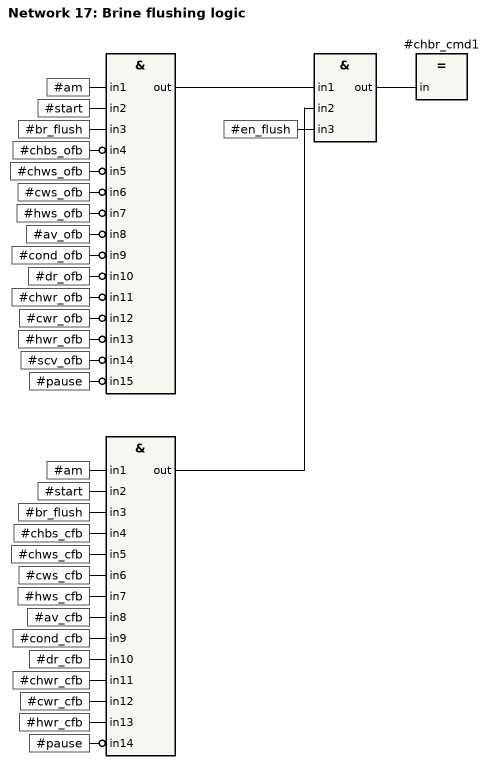
   #chbr_cmd1 := #am AND #start AND #br_flush AND NOT #chbs_ofb AND NOT #chws_ofb AND NOT #cws_ofb AND NOT #hws_ofb AND NOT #av_ofb AND NOT #cond_ofb AND NOT #dr_ofb AND NOT #chwr_ofb AND NOT #cwr_ofb AND NOT #hwr_ofb AND NOT #scv_ofb AND NOT #pause AND #am AND #start AND #br_flush AND #chbs_cfb AND #chws_cfb AND #cws_cfb AND #hws_cfb AND #av_cfb AND #cond_cfb AND #dr_cfb AND #chwr_cfb AND #cwr_cfb AND #hwr_cfb AND NOT #pause AND #en_flush;
END_REGION

REGION Network 18: Steam flushing logic
   // Steam flushing logic
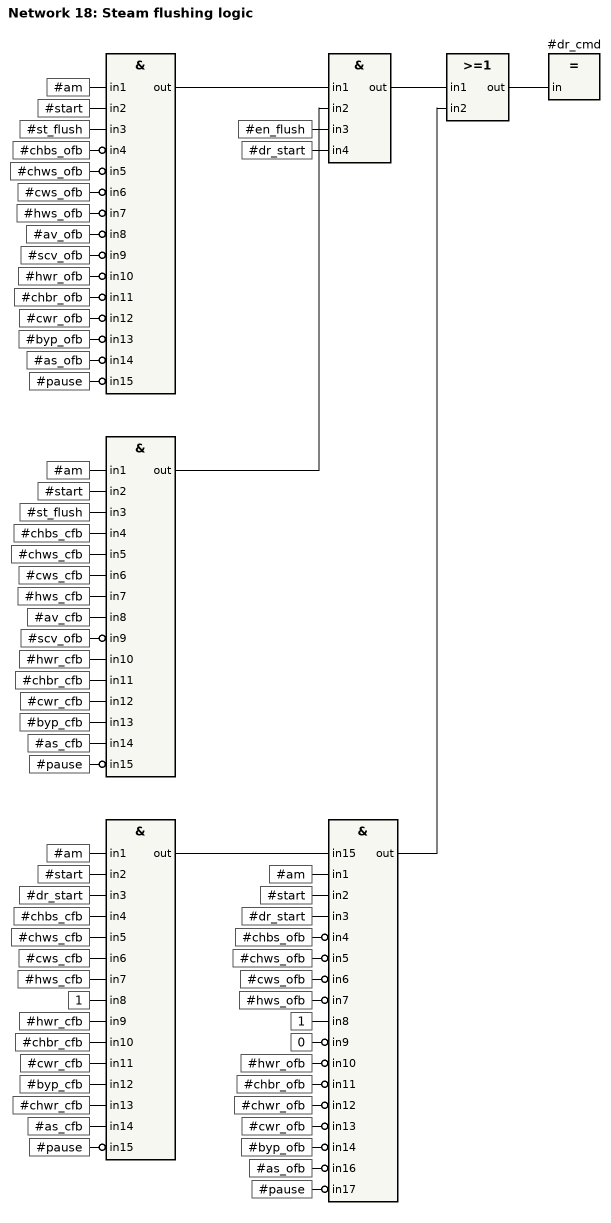
   #dr_cmd := (#am AND #start AND #st_flush AND NOT #chbs_ofb AND NOT #chws_ofb AND NOT #cws_ofb AND NOT #hws_ofb AND NOT #av_ofb AND NOT #scv_ofb AND NOT #hwr_ofb AND NOT #chbr_ofb AND NOT #cwr_ofb AND NOT #byp_ofb AND NOT #as_ofb AND NOT #pause AND #am AND #start AND #st_flush AND #chbs_cfb AND #chws_cfb AND #cws_cfb AND #hws_cfb AND #av_cfb AND NOT #scv_ofb AND #hwr_cfb AND #chbr_cfb AND #cwr_cfb AND #byp_cfb AND #as_cfb AND NOT #pause AND #en_flush AND #dr_start) OR (#am AND #start AND #dr_start AND #chbs_cfb AND #chws_cfb AND #cws_cfb AND #hws_cfb AND 1 AND #hwr_cfb AND #chbr_cfb AND #cwr_cfb AND #byp_cfb AND #chwr_cfb AND #as_cfb AND NOT #pause AND #am AND #start AND #dr_start AND NOT #chbs_ofb AND NOT #chws_ofb AND NOT #cws_ofb AND NOT #hws_ofb AND 1 AND NOT 0 AND NOT #hwr_ofb AND NOT #chbr_ofb AND NOT #chwr_ofb AND NOT #cwr_ofb AND NOT #byp_ofb AND NOT #as_ofb AND NOT #pause);
END_REGION

REGION Network 19: chw flushing logic
   // chw flushing logic
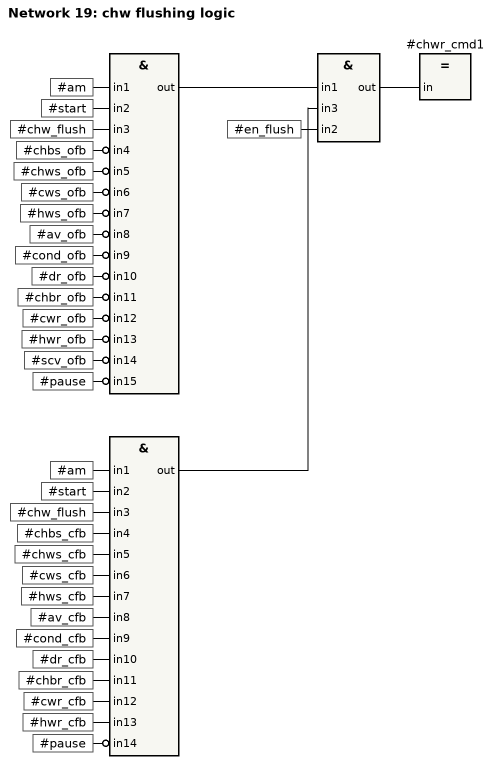
   #chwr_cmd1 := #am AND #start AND #chw_flush AND NOT #chbs_ofb AND NOT #chws_ofb AND NOT #cws_ofb AND NOT #hws_ofb AND NOT #av_ofb AND NOT #cond_ofb AND NOT #dr_ofb AND NOT #chbr_ofb AND NOT #cwr_ofb AND NOT #hwr_ofb AND NOT #scv_ofb AND NOT #pause AND #am AND #start AND #chw_flush AND #chbs_cfb AND #chws_cfb AND #cws_cfb AND #hws_cfb AND #av_cfb AND #cond_cfb AND #dr_cfb AND #chbr_cfb AND #cwr_cfb AND #hwr_cfb AND NOT #pause AND #en_flush;
END_REGION

REGION Network 20: air supply and bypass open logic
   // air supply and bypass open logic
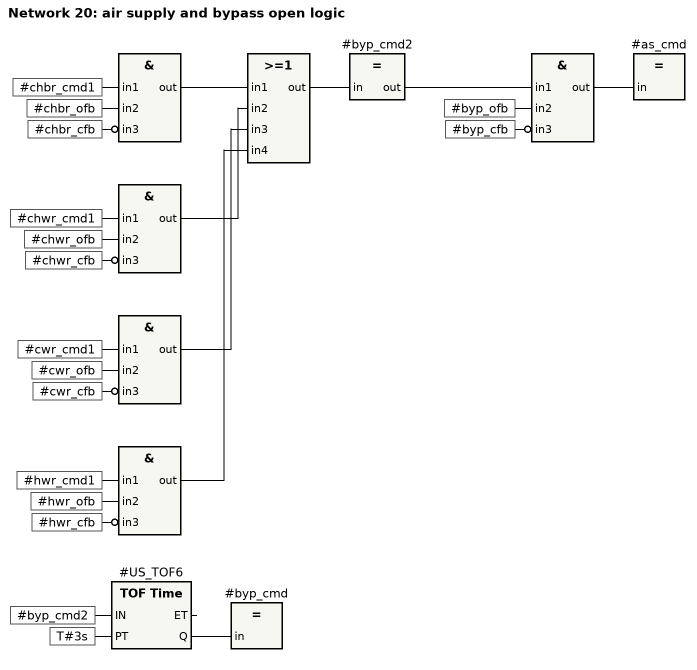
   #byp_cmd2 := (#chbr_cmd1 AND #chbr_ofb AND NOT #chbr_cfb) OR (#chwr_cmd1 AND #chwr_ofb AND NOT #chwr_cfb) OR (#cwr_cmd1 AND #cwr_ofb AND NOT #cwr_cfb) OR (#hwr_cmd1 AND #hwr_ofb AND NOT #hwr_cfb);
   #as_cmd := #byp_cmd2 AND #byp_ofb AND NOT #byp_cfb;
   #US_TOF6(IN := #byp_cmd2, PT := T#3s);   // TOF
   #byp_cmd := #US_TOF6.Q;
END_REGION

REGION Network 21: CW flushing logic
   // CW flushing logic
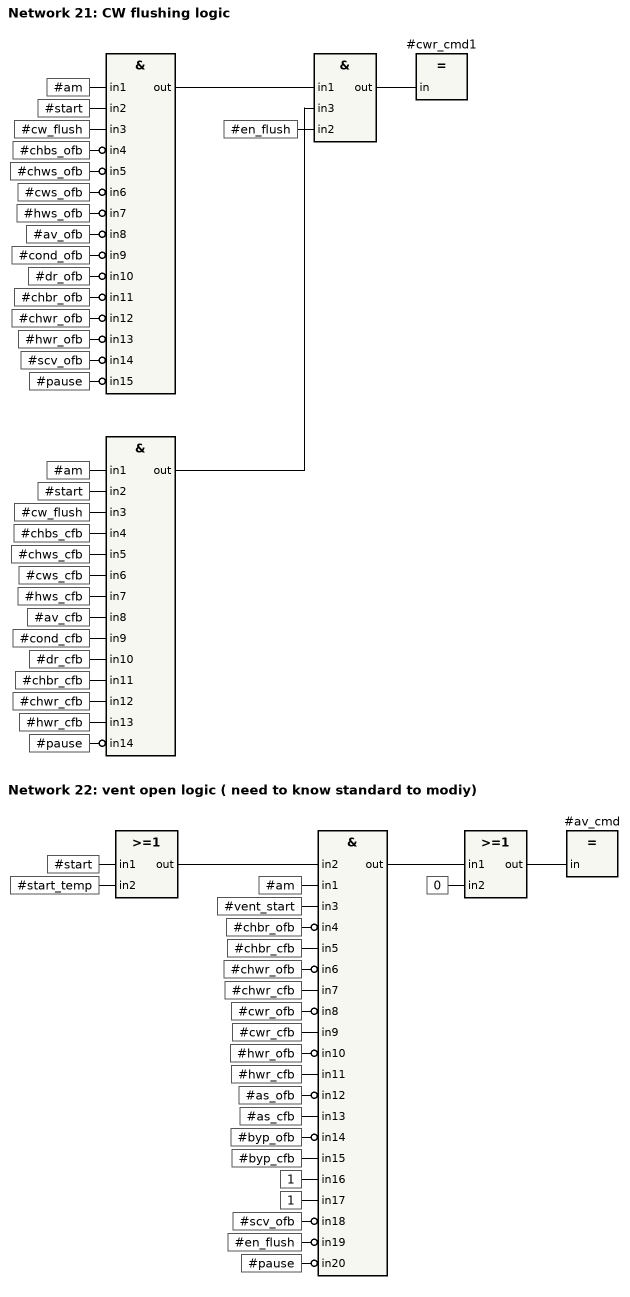
   #cwr_cmd1 := #am AND #start AND #cw_flush AND NOT #chbs_ofb AND NOT #chws_ofb AND NOT #cws_ofb AND NOT #hws_ofb AND NOT #av_ofb AND NOT #cond_ofb AND NOT #dr_ofb AND NOT #chbr_ofb AND NOT #chwr_ofb AND NOT #hwr_ofb AND NOT #scv_ofb AND NOT #pause AND #am AND #start AND #cw_flush AND #chbs_cfb AND #chws_cfb AND #cws_cfb AND #hws_cfb AND #av_cfb AND #cond_cfb AND #dr_cfb AND #chbr_cfb AND #chwr_cfb AND #hwr_cfb AND NOT #pause AND #en_flush;
END_REGION

REGION Network 22: vent open logic ( need to know standard to modiy)
   // vent open logic
   #av_cmd := ((#start OR #start_temp) AND #am AND #vent_start AND NOT #chbr_ofb AND #chbr_cfb AND NOT #chwr_ofb AND #chwr_cfb AND NOT #cwr_ofb AND #cwr_cfb AND NOT #hwr_ofb AND #hwr_cfb AND NOT #as_ofb AND #as_cfb AND NOT #byp_ofb AND #byp_cfb AND 1 AND 1 AND NOT #scv_ofb AND NOT #en_flush AND NOT #pause) OR 0;
END_REGION

REGION Network 23: hw flushing logic
   // hw flushing logic
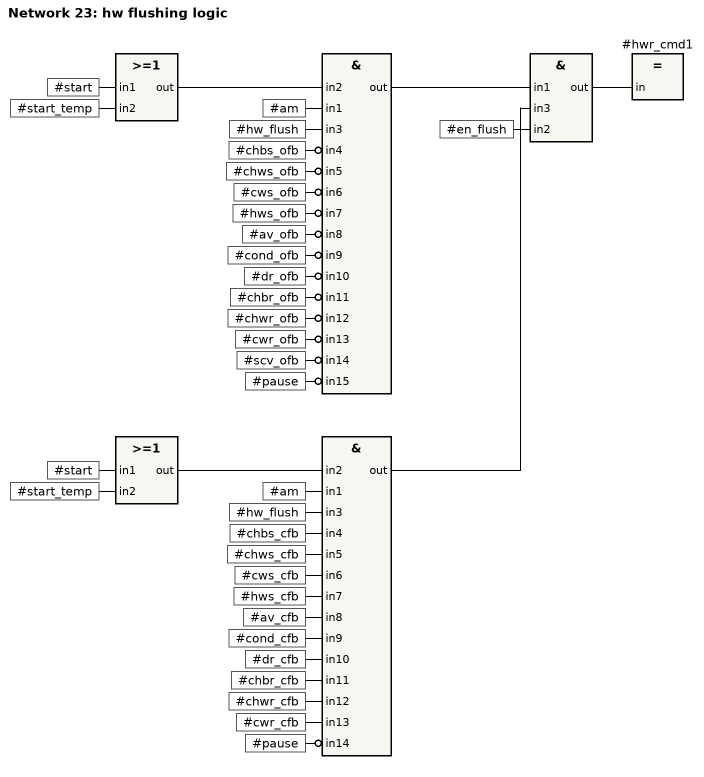
   #hwr_cmd1 := (#start OR #start_temp) AND #am AND #hw_flush AND NOT #chbs_ofb AND NOT #chws_ofb AND NOT #cws_ofb AND NOT #hws_ofb AND NOT #av_ofb AND NOT #cond_ofb AND NOT #dr_ofb AND NOT #chbr_ofb AND NOT #chwr_ofb AND NOT #cwr_ofb AND NOT #scv_ofb AND NOT #pause AND (#start OR #start_temp) AND #am AND #hw_flush AND #chbs_cfb AND #chws_cfb AND #cws_cfb AND #hws_cfb AND #av_cfb AND #cond_cfb AND #dr_cfb AND #chbr_cfb AND #chwr_cfb AND #cwr_cfb AND NOT #pause AND #en_flush;
END_REGION
END_FUNCTION_BLOCK

FUNCTION "Word_to_Bit" : Void
{ S7_Optimized_Access := 'TRUE' }
VERSION : 0.1
   VAR_INPUT 
      "word" : Word;
   END_VAR

   VAR_OUTPUT 
      Bit0 : Bool;
      Bit1 : Bool;
      Bit2 : Bool;
      Bit3 : Bool;
      Bit4 : Bool;
      Bit5 : Bool;
      Bit6 : Bool;
      Bit7 : Bool;
      Bit8 : Bool;
      Bit9 : Bool;
      Bit10 : Bool;
      Bit11 : Bool;
      Bit12 : Bool;
      Bit13 : Bool;
      Bit14 : Bool;
      Bit15 : Bool;
   END_VAR


BEGIN
	#Bit0 := #"word".%X0;
	#Bit1 := #"word".%X1;
	#Bit2 := #"word".%X2;
	#Bit3 := #"word".%X3;
	#Bit4 := #"word".%X4;
	#Bit5 := #"word".%X5;
	#Bit6 := #"word".%X6;
	#Bit7 := #"word".%X7;
	#Bit8 := #"word".%X8;
	#Bit9 := #"word".%X9;
	#Bit10 := #"word".%X10;
	#Bit11 := #"word".%X11;
	#Bit12 := #"word".%X12;
	#Bit13 := #"word".%X13;
	#Bit14 := #"word".%X14;
	#Bit15 := #"word".%X15;
END_FUNCTION

FUNCTION "Bit_to_Word" : Void
{ S7_Optimized_Access := 'TRUE' }
VERSION : 0.1
   VAR_INPUT 
      Bit0 : Bool;
      Bit1 : Bool;
      Bit2 : Bool;
      Bit3 : Bool;
      Bit4 : Bool;
      Bit5 : Bool;
      Bit6 : Bool;
      Bit7 : Bool;
      Bit8 : Bool;
      Bit9 : Bool;
      Bit10 : Bool;
      Bit11 : Bool;
      Bit12 : Bool;
      Bit13 : Bool;
      Bit14 : Bool;
      Bit15 : Bool;
   END_VAR

   VAR_OUTPUT 
      "word" : Word;
   END_VAR


BEGIN
	#"word".%X0 := #Bit0;
	#"word".%X1 := #Bit1;
	#"word".%X2 := #Bit2;
	#"word".%X3 := #Bit3;
	#"word".%X4 := #Bit4;
	#"word".%X5 := #Bit5;
	#"word".%X6 := #Bit6;
	#"word".%X7 := #Bit7;
	#"word".%X8 := #Bit8;
	#"word".%X9 := #Bit9;
	#"word".%X10 := #Bit10;
	#"word".%X11 := #Bit11;
	#"word".%X12 := #Bit12;
	#"word".%X13 := #Bit13;
	#"word".%X14 := #Bit14;
	#"word".%X15:= #Bit15;
	
END_FUNCTION

ORGANIZATION_BLOCK "Cyclic interrupt"   // OB31, FBD, CyclicInterrupt
{ S7_Optimized_Access := 'TRUE' }
VERSION : 0.1
// stored: AutoNumber true, IsIECCheckEnabled false, SetENOAutomatically false
   VAR_INPUT
      Initial_Call : Bool;   // Initial call of this OB
      Event_Count : Int;   // Events discarded
   END_VAR
BEGIN

REGION Network 1
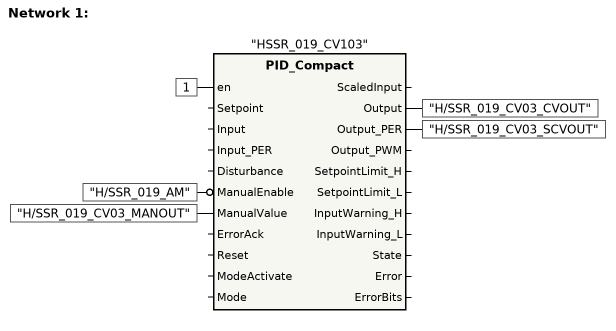
   IF 1 THEN
       "HSSR_019_CV103"(ManualEnable := NOT "H/SSR_019_AM",   // PID_Compact
                        ManualValue := "H/SSR_019_CV03_MANOUT",
                        Output => "H/SSR_019_CV03_CVOUT",
                        Output_PER => "H/SSR_019_CV03_SCVOUT");
   END_IF;
END_REGION
END_ORGANIZATION_BLOCK

ORGANIZATION_BLOCK "Main"   // OB123, FBD, ProgramCycle
TITLE = "Main Program Sweep (Cycle)"
{ S7_Optimized_Access := 'TRUE' }
VERSION : 0.1
// stored: AutoNumber true, IsIECCheckEnabled false, SetENOAutomatically false
   VAR_INPUT
      Initial_Call : Bool;   // Initial call of this OB
      Remanence : Bool;   // =True, if remanent data are available
   END_VAR
BEGIN

REGION Network 1 (SCL): HSSR_019 SOURCE SELECTION

   "Source_select_H/SSR_019_DB".START := "H/SSR_019_START";
   "Source_select_H/SSR_019_DB".SP := "H/SSR_019_SP";
   "Source_select_H/SSR_019_DB".PV := "H/SSR_019_TT01_PV";
   "Source_select_H/SSR_019_DB".COUNTER_SP := "H/SSR_019_ALERT_SP";
   "Source_select_H/SSR_019_DB".CHW_CT_SP := "H/SSR_019_CHBr_RT_SP";
   "Source_select_H/SSR_019_DB".CT_HW_SP := "H/SSR_019_RT_HW_SP";
   "Source_select_H/SSR_019_DB".HW_STEAM_SP := "H/SSR_019_HW_STEAM_SP";
   "Source_select_H/SSR_019_DB".CT_CHW_SP := "H/SSR_019_RT_CHBr_SP";

   "H/SSR_019_SOURCE_SEL" := "Source_select_H/SSR_019_DB".SOURCE_SEL;
END_REGION

REGION Network 2 (SCL): HSSR_019 UTILITY PID

   "Utility_PID_DB".AM := "H/SSR_019_AM";
   "Utility_PID_DB".START := "H/SSR_019_START";
   "Utility_PID_DB".SP := "H/SSR_019_SP";
   "Utility_PID_DB".PV := "H/SSR_019_TT01_PV";
   "Utility_PID_DB".TIME := "H/SSR_019_TIME_SP";
   "Utility_PID_DB".P := "H/SSR_019_KP";
   "Utility_PID_DB".I := "H/SSR_019_TI";
   "Utility_PID_DB".JAC_IN := "H/SSR_019_TT02_PV";
   "Utility_PID_DB".SOURCE_SEL := "Source_select_H/SSR_019_DB".SOURCE_SEL;
   "Utility_PID_DB".MAN_OUT := "H/SSR_019_CV02_MANOUT";
   "Utility_PID_DB".STEAM_MAN_OUT := "H/SSR_019_CV01_MANOUT";
   "Utility_PID_DB".AIR_XV_OPN := "H/SSR_019_XV10_CMD";
   "Utility_PID_DB".BYP_XV_OPN := "H/SSR_019_XV05_CMD";
   "Utility_PID_DB".VENT_OPN := "H/SSR_019_XV06_CMD";
   "Utility_PID_DB".CONDENSATE_XV_OPN := "H/SSR_019_XV12_CMD";
   "Utility_PID_DB".DRAIN_XV_OPN := "H/SSR_019_XV13_CMD";
   "Utility_PID_DB".CONTROL_MODE := 1;

   "H/SSR_019_START_PV" := "Utility_PID_DB".START_PV;
   "H/SSR_019_CV02_SCVOUT" := "Utility_PID_DB".SCVOUT;
   "H/SSR_019_CV02_CVOUT" := "Utility_PID_DB".CVOUT;
   "H/SSR_019_CV01_SCVOUT" := "Utility_PID_DB".STEAM_SCVOUT;
   "H/SSR_019_CV01_CVOUT" := "Utility_PID_DB".STEAM_CVOUT;
   "H/SSR_019_RUN_MIN" := "Utility_PID_DB".RUN_MIN;
END_REGION

REGION Network 3 (SCL): HSSR_019 UTILITY SELECTION

   "Utility_selection_DB".utl_type :=  "Source_select_H/SSR_019_DB".SOURCE_SEL;
   "Utility_selection_DB".chws_cfb :="SIM_VALVE"."H/SSR_019_XV01_CLOSEFB" ;
   "Utility_selection_DB".chws_ofb := "SIM_VALVE"."H/SSR_019_XV01_OPENFB";
   "Utility_selection_DB".cws_cfb := "SIM_VALVE"."H/SSR_019_XV02_CLOSEFB";
   "Utility_selection_DB".cws_ofb := "SIM_VALVE"."H/SSR_019_XV02_OPENFB";
   "Utility_selection_DB".hws_cfb := "SIM_VALVE"."H/SSR_019_XV03_CLOSEFB";
   "Utility_selection_DB".hws_ofb := "SIM_VALVE"."H/SSR_019_XV03_OPENFB";
   "Utility_selection_DB".chwr_cfb := "SIM_VALVE"."H/SSR_019_XV07_CLOSEFB";
   "Utility_selection_DB".chwr_ofb := "SIM_VALVE"."H/SSR_019_XV07_OPENFB";
   "Utility_selection_DB".cwr_cfb := "SIM_VALVE"."H/SSR_019_XV08_CLOSEFB";
   "Utility_selection_DB".cwr_ofb := "SIM_VALVE"."H/SSR_019_XV08_OPENFB";
   "Utility_selection_DB".hwr_cfb := "SIM_VALVE"."H/SSR_019_XV09_CLOSEFB";
   "Utility_selection_DB".hwr_ofb := "SIM_VALVE"."H/SSR_019_XV09_OPENFB";
   "Utility_selection_DB".scv_ofb := "SIM_VALVE"."H/SSR_019_XV11_OPENFB";
   "Utility_selection_DB".cond_cfb := "SIM_VALVE"."H/SSR_019_XV12_CLOSEFB";
   "Utility_selection_DB".cond_ofb := "SIM_VALVE"."H/SSR_019_XV12_OPENFB";
   "Utility_selection_DB".dr_cfb := "SIM_VALVE"."H/SSR_019_XV13_CLOSEFB";
   "Utility_selection_DB".dr_ofb := "SIM_VALVE"."H/SSR_019_XV13_OPENFB";
   "Utility_selection_DB".as_cfb := "SIM_VALVE"."H/SSR_019_XV10_CLOSEFB";
   "Utility_selection_DB".as_ofb := "SIM_VALVE"."H/SSR_019_XV10_OPENFB";
   "Utility_selection_DB".av_cfb := "SIM_VALVE"."H/SSR_019_XV06_CLOSEFB";
   "Utility_selection_DB".av_ofb := "SIM_VALVE"."H/SSR_019_XV06_OPENFB";
   "Utility_selection_DB".utl_bit := "H/SSR_019_START";
   "Utility_selection_DB".control.%X1 := "H/SSR_019_AM";
   "Utility_selection_DB".control.%X2 := "H/SSR_019_START";
   "Utility_selection_DB".times[0] := "H/SSR_019_FLUSH_TIME_SP";
   "Utility_selection_DB".times[1] := "H/SSR_019_VENT_TIME_SP";
   "Utility_selection_DB".times[2] := "H/SSR_019_CONDENSATE_TIME_SP";
   "Utility_selection_DB".control.%X0   := "H/SSR_019_HOLD";
   "Utility_selection_DB".control.%X6 := "H/SSR_019_EMSTOP";
   "Utility_selection_DB".byp_cfb := "SIM_VALVE"."H/SSR_019_XV05_CLOSEFB";
   "Utility_selection_DB".byp_ofb := "SIM_VALVE"."H/SSR_019_XV05_OPENFB";
   "H/SSR_019_XV01_CMD" := "Utility_selection_DB".chws_cmd;
   "H/SSR_019_XV02_CMD" := "Utility_selection_DB".cws_cmd;
   "H/SSR_019_XV03_CMD" := "Utility_selection_DB".hws_cmd;
   "H/SSR_019_XV07_CMD" := "Utility_selection_DB".chwr_cmd;
   "H/SSR_019_XV08_CMD" := "Utility_selection_DB".cwr_cmd;
   "H/SSR_019_XV09_CMD" := "Utility_selection_DB".hwr_cmd;
   "H/SSR_019_XV11_CMD" := "Utility_selection_DB".scv_cmd;
   "H/SSR_019_XV12_CMD" := "Utility_selection_DB".cond_cmd;
   "H/SSR_019_XV13_CMD" := "Utility_selection_DB".dr_cmd;
   "H/SSR_019_XV10_CMD" := "Utility_selection_DB".as_cmd;
   "H/SSR_019_XV05_CMD" := "Utility_selection_DB".byp_cmd;
   "H/SSR_019_XV06_CMD" := "Utility_selection_DB".av_cmd;
   "H/SSR_019_FLUSH_RUN_TIME" := "Utility_selection_DB".flush_time;
   "H/SSR_019_CONDENSATE_RUN_TIME" := "Utility_selection_DB".drine_time;
   "H/SSR_019_VENT_RUN_TIME" := "Utility_selection_DB".vent_time;
   "H/SSR_019_Flush_CMP" := "Utility_selection_DB".status.%X2;
   "H/SSR_019_Vent_CMP" := "Utility_selection_DB".status.%X3;
   "H/SSR_019_Cond_CMP" := "Utility_selection_DB".status.%X4;
END_REGION

REGION Network 4: HSSR_019_Pre checks
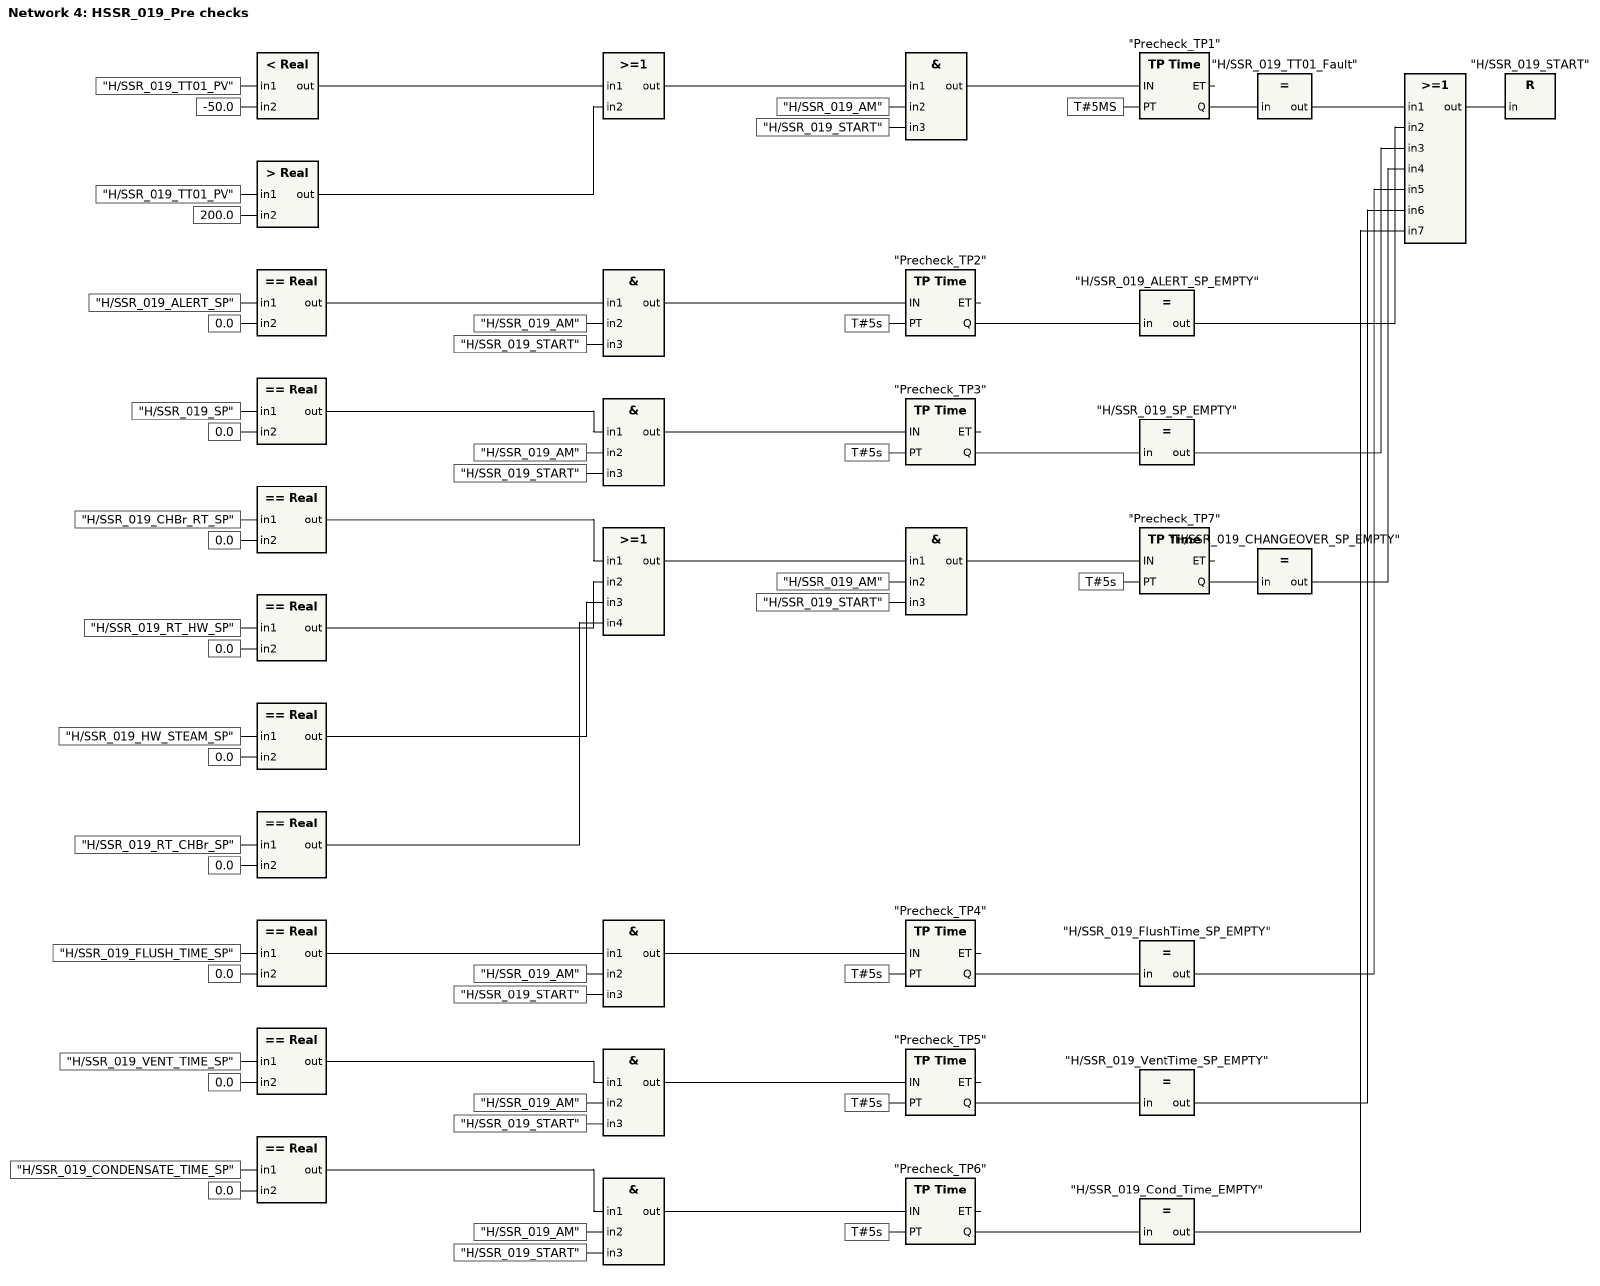
   "Precheck_TP1".TP(IN := (("H/SSR_019_TT01_PV" < (-50.0)) OR ("H/SSR_019_TT01_PV" > 200.0)) AND "H/SSR_019_AM" AND "H/SSR_019_START",
                     PT := T#5MS);
   "H/SSR_019_TT01_Fault" := "Precheck_TP1".Q;
   "Precheck_TP2".TP(IN := ("H/SSR_019_ALERT_SP" = 0.0) AND "H/SSR_019_AM" AND "H/SSR_019_START", PT := T#5s);
   "H/SSR_019_ALERT_SP_EMPTY" := "Precheck_TP2".Q;
   "Precheck_TP3".TP(IN := ("H/SSR_019_SP" = 0.0) AND "H/SSR_019_AM" AND "H/SSR_019_START", PT := T#5s);
   "H/SSR_019_SP_EMPTY" := "Precheck_TP3".Q;
   "Precheck_TP7".TP(IN := (("H/SSR_019_CHBr_RT_SP" = 0.0) OR ("H/SSR_019_RT_HW_SP" = 0.0) OR ("H/SSR_019_HW_STEAM_SP" = 0.0) OR ("H/SSR_019_RT_CHBr_SP" = 0.0)) AND "H/SSR_019_AM" AND "H/SSR_019_START",
                     PT := T#5s);
   "H/SSR_019_CHANGEOVER_SP_EMPTY" := "Precheck_TP7".Q;
   "Precheck_TP4".TP(IN := ("H/SSR_019_FLUSH_TIME_SP" = 0.0) AND "H/SSR_019_AM" AND "H/SSR_019_START",
                     PT := T#5s);
   "H/SSR_019_FlushTime_SP_EMPTY" := "Precheck_TP4".Q;
   "Precheck_TP5".TP(IN := ("H/SSR_019_VENT_TIME_SP" = 0.0) AND "H/SSR_019_AM" AND "H/SSR_019_START",
                     PT := T#5s);
   "H/SSR_019_VentTime_SP_EMPTY" := "Precheck_TP5".Q;
   "Precheck_TP6".TP(IN := ("H/SSR_019_CONDENSATE_TIME_SP" = 0.0) AND "H/SSR_019_AM" AND "H/SSR_019_START",
                     PT := T#5s);
   "H/SSR_019_Cond_Time_EMPTY" := "Precheck_TP6".Q;
   IF "Precheck_TP1".Q OR "Precheck_TP2".Q OR "Precheck_TP3".Q OR "Precheck_TP7".Q OR "Precheck_TP4".Q OR "Precheck_TP5".Q OR "Precheck_TP6".Q THEN
       "H/SSR_019_START" := FALSE;
   END_IF;
END_REGION

REGION Network 5: H/SSR_019Valves
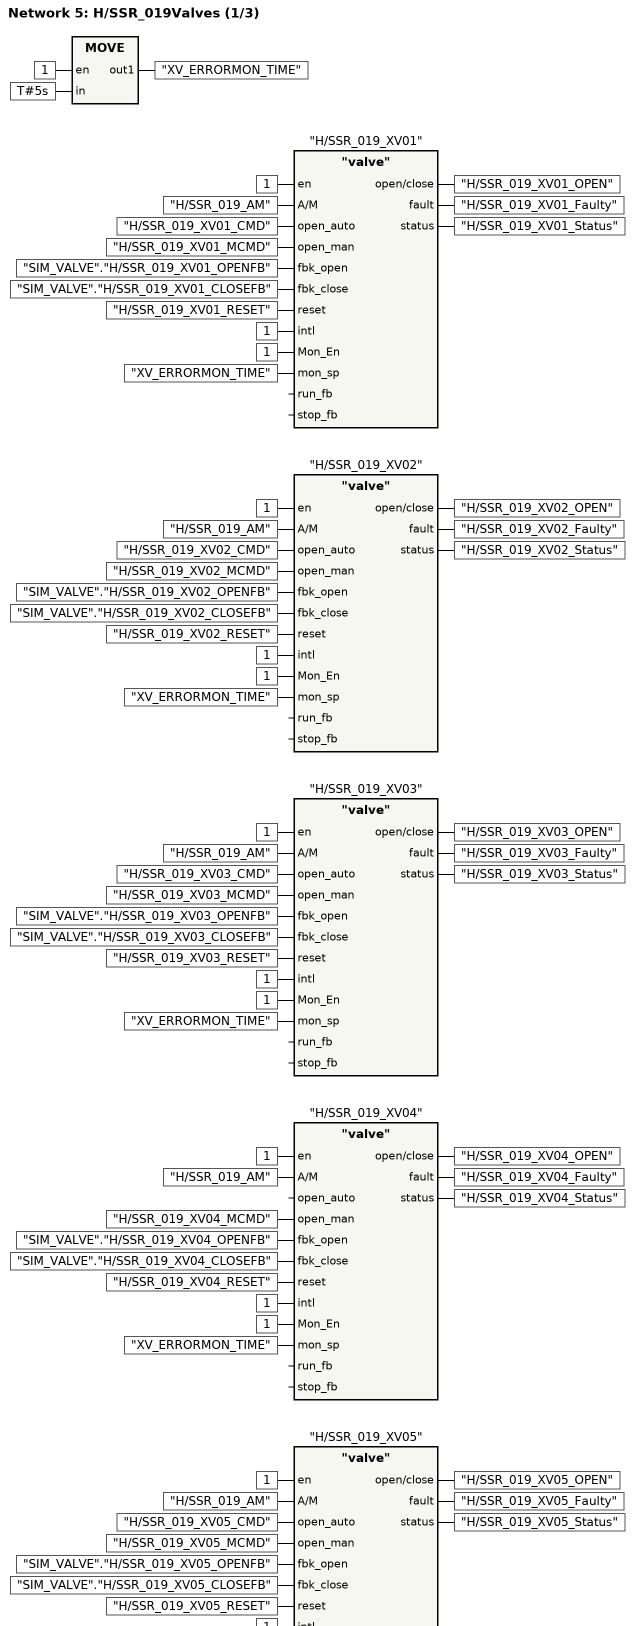
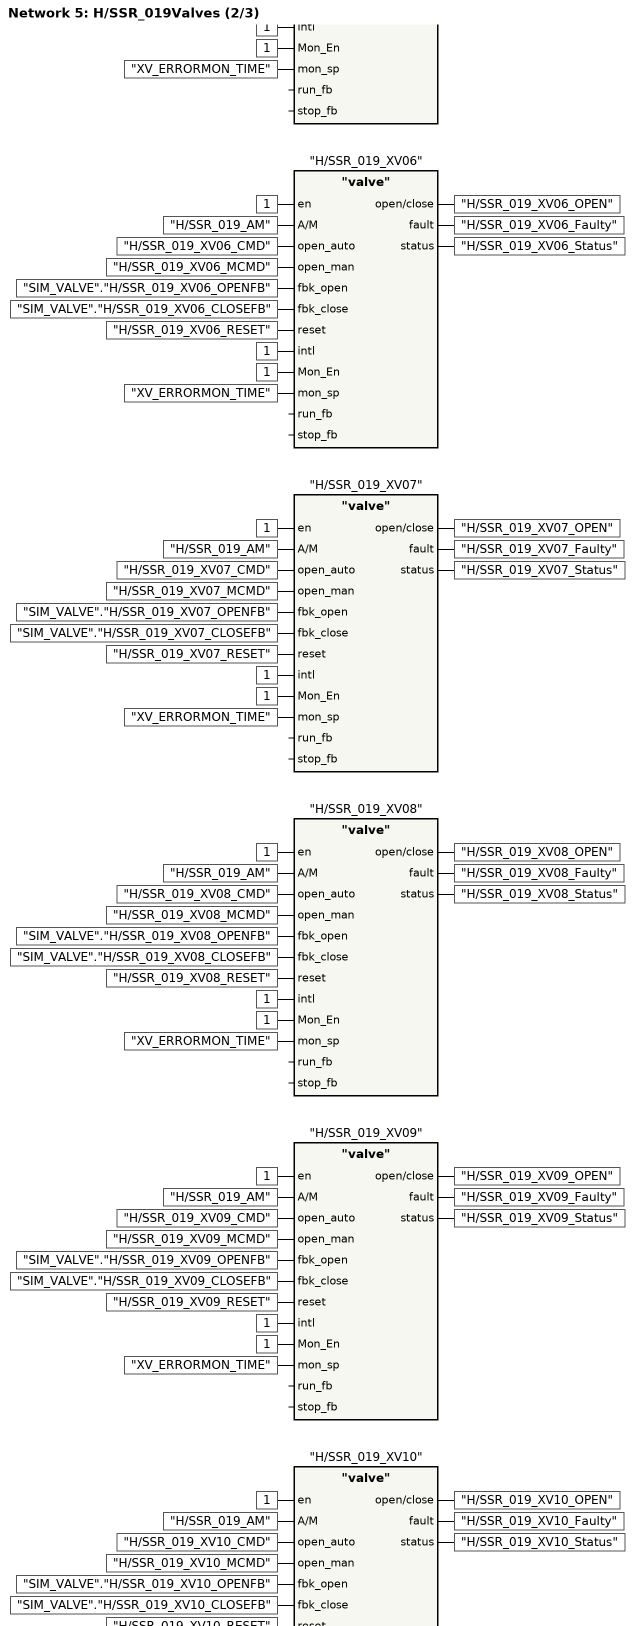
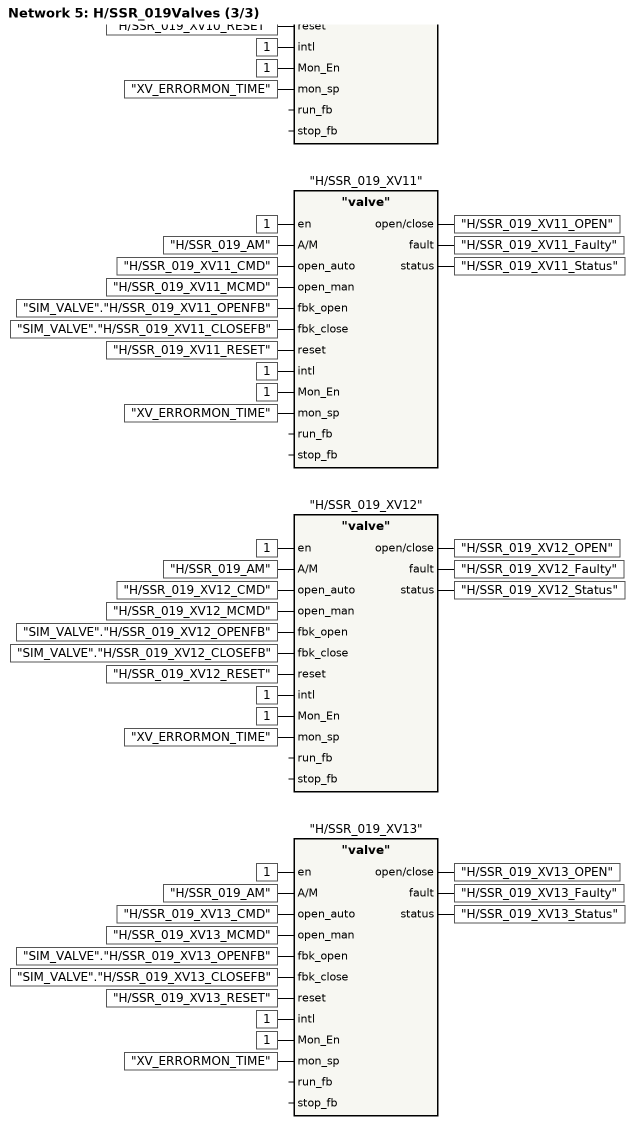
   IF 1 THEN
       "XV_ERRORMON_TIME" := T#5s;
       "H/SSR_019_XV01"("A/M" := "H/SSR_019_AM",   // "valve"
                        open_auto := "H/SSR_019_XV01_CMD",
                        open_man := "H/SSR_019_XV01_MCMD",
                        fbk_open := "SIM_VALVE"."H/SSR_019_XV01_OPENFB",
                        fbk_close := "SIM_VALVE"."H/SSR_019_XV01_CLOSEFB",
                        reset := "H/SSR_019_XV01_RESET",
                        intl := 1,
                        Mon_En := 1,
                        mon_sp := "XV_ERRORMON_TIME",
                        "open/close" => "H/SSR_019_XV01_OPEN",
                        fault => "H/SSR_019_XV01_Faulty",
                        status => "H/SSR_019_XV01_Status");
       "H/SSR_019_XV02"("A/M" := "H/SSR_019_AM",   // "valve"
                        open_auto := "H/SSR_019_XV02_CMD",
                        open_man := "H/SSR_019_XV02_MCMD",
                        fbk_open := "SIM_VALVE"."H/SSR_019_XV02_OPENFB",
                        fbk_close := "SIM_VALVE"."H/SSR_019_XV02_CLOSEFB",
                        reset := "H/SSR_019_XV02_RESET",
                        intl := 1,
                        Mon_En := 1,
                        mon_sp := "XV_ERRORMON_TIME",
                        "open/close" => "H/SSR_019_XV02_OPEN",
                        fault => "H/SSR_019_XV02_Faulty",
                        status => "H/SSR_019_XV02_Status");
       "H/SSR_019_XV03"("A/M" := "H/SSR_019_AM",   // "valve"
                        open_auto := "H/SSR_019_XV03_CMD",
                        open_man := "H/SSR_019_XV03_MCMD",
                        fbk_open := "SIM_VALVE"."H/SSR_019_XV03_OPENFB",
                        fbk_close := "SIM_VALVE"."H/SSR_019_XV03_CLOSEFB",
                        reset := "H/SSR_019_XV03_RESET",
                        intl := 1,
                        Mon_En := 1,
                        mon_sp := "XV_ERRORMON_TIME",
                        "open/close" => "H/SSR_019_XV03_OPEN",
                        fault => "H/SSR_019_XV03_Faulty",
                        status => "H/SSR_019_XV03_Status");
       "H/SSR_019_XV04"("A/M" := "H/SSR_019_AM",   // "valve"
                        open_man := "H/SSR_019_XV04_MCMD",
                        fbk_open := "SIM_VALVE"."H/SSR_019_XV04_OPENFB",
                        fbk_close := "SIM_VALVE"."H/SSR_019_XV04_CLOSEFB",
                        reset := "H/SSR_019_XV04_RESET",
                        intl := 1,
                        Mon_En := 1,
                        mon_sp := "XV_ERRORMON_TIME",
                        "open/close" => "H/SSR_019_XV04_OPEN",
                        fault => "H/SSR_019_XV04_Faulty",
                        status => "H/SSR_019_XV04_Status");
       "H/SSR_019_XV05"("A/M" := "H/SSR_019_AM",   // "valve"
                        open_auto := "H/SSR_019_XV05_CMD",
                        open_man := "H/SSR_019_XV05_MCMD",
                        fbk_open := "SIM_VALVE"."H/SSR_019_XV05_OPENFB",
                        fbk_close := "SIM_VALVE"."H/SSR_019_XV05_CLOSEFB",
                        reset := "H/SSR_019_XV05_RESET",
                        intl := 1,
                        Mon_En := 1,
                        mon_sp := "XV_ERRORMON_TIME",
                        "open/close" => "H/SSR_019_XV05_OPEN",
                        fault => "H/SSR_019_XV05_Faulty",
                        status => "H/SSR_019_XV05_Status");
       "H/SSR_019_XV06"("A/M" := "H/SSR_019_AM",   // "valve"
                        open_auto := "H/SSR_019_XV06_CMD",
                        open_man := "H/SSR_019_XV06_MCMD",
                        fbk_open := "SIM_VALVE"."H/SSR_019_XV06_OPENFB",
                        fbk_close := "SIM_VALVE"."H/SSR_019_XV06_CLOSEFB",
                        reset := "H/SSR_019_XV06_RESET",
                        intl := 1,
                        Mon_En := 1,
                        mon_sp := "XV_ERRORMON_TIME",
                        "open/close" => "H/SSR_019_XV06_OPEN",
                        fault => "H/SSR_019_XV06_Faulty",
                        status => "H/SSR_019_XV06_Status");
       "H/SSR_019_XV07"("A/M" := "H/SSR_019_AM",   // "valve"
                        open_auto := "H/SSR_019_XV07_CMD",
                        open_man := "H/SSR_019_XV07_MCMD",
                        fbk_open := "SIM_VALVE"."H/SSR_019_XV07_OPENFB",
                        fbk_close := "SIM_VALVE"."H/SSR_019_XV07_CLOSEFB",
                        reset := "H/SSR_019_XV07_RESET",
                        intl := 1,
                        Mon_En := 1,
                        mon_sp := "XV_ERRORMON_TIME",
                        "open/close" => "H/SSR_019_XV07_OPEN",
                        fault => "H/SSR_019_XV07_Faulty",
                        status => "H/SSR_019_XV07_Status");
       "H/SSR_019_XV08"("A/M" := "H/SSR_019_AM",   // "valve"
                        open_auto := "H/SSR_019_XV08_CMD",
                        open_man := "H/SSR_019_XV08_MCMD",
                        fbk_open := "SIM_VALVE"."H/SSR_019_XV08_OPENFB",
                        fbk_close := "SIM_VALVE"."H/SSR_019_XV08_CLOSEFB",
                        reset := "H/SSR_019_XV08_RESET",
                        intl := 1,
                        Mon_En := 1,
                        mon_sp := "XV_ERRORMON_TIME",
                        "open/close" => "H/SSR_019_XV08_OPEN",
                        fault => "H/SSR_019_XV08_Faulty",
                        status => "H/SSR_019_XV08_Status");
       "H/SSR_019_XV09"("A/M" := "H/SSR_019_AM",   // "valve"
                        open_auto := "H/SSR_019_XV09_CMD",
                        open_man := "H/SSR_019_XV09_MCMD",
                        fbk_open := "SIM_VALVE"."H/SSR_019_XV09_OPENFB",
                        fbk_close := "SIM_VALVE"."H/SSR_019_XV09_CLOSEFB",
                        reset := "H/SSR_019_XV09_RESET",
                        intl := 1,
                        Mon_En := 1,
                        mon_sp := "XV_ERRORMON_TIME",
                        "open/close" => "H/SSR_019_XV09_OPEN",
                        fault => "H/SSR_019_XV09_Faulty",
                        status => "H/SSR_019_XV09_Status");
       "H/SSR_019_XV10"("A/M" := "H/SSR_019_AM",   // "valve"
                        open_auto := "H/SSR_019_XV10_CMD",
                        open_man := "H/SSR_019_XV10_MCMD",
                        fbk_open := "SIM_VALVE"."H/SSR_019_XV10_OPENFB",
                        fbk_close := "SIM_VALVE"."H/SSR_019_XV10_CLOSEFB",
                        reset := "H/SSR_019_XV10_RESET",
                        intl := 1,
                        Mon_En := 1,
                        mon_sp := "XV_ERRORMON_TIME",
                        "open/close" => "H/SSR_019_XV10_OPEN",
                        fault => "H/SSR_019_XV10_Faulty",
                        status => "H/SSR_019_XV10_Status");
       "H/SSR_019_XV11"("A/M" := "H/SSR_019_AM",   // "valve"
                        open_auto := "H/SSR_019_XV11_CMD",
                        open_man := "H/SSR_019_XV11_MCMD",
                        fbk_open := "SIM_VALVE"."H/SSR_019_XV11_OPENFB",
                        fbk_close := "SIM_VALVE"."H/SSR_019_XV11_CLOSEFB",
                        reset := "H/SSR_019_XV11_RESET",
                        intl := 1,
                        Mon_En := 1,
                        mon_sp := "XV_ERRORMON_TIME",
                        "open/close" => "H/SSR_019_XV11_OPEN",
                        fault => "H/SSR_019_XV11_Faulty",
                        status => "H/SSR_019_XV11_Status");
       "H/SSR_019_XV12"("A/M" := "H/SSR_019_AM",   // "valve"
                        open_auto := "H/SSR_019_XV12_CMD",
                        open_man := "H/SSR_019_XV12_MCMD",
                        fbk_open := "SIM_VALVE"."H/SSR_019_XV12_OPENFB",
                        fbk_close := "SIM_VALVE"."H/SSR_019_XV12_CLOSEFB",
                        reset := "H/SSR_019_XV12_RESET",
                        intl := 1,
                        Mon_En := 1,
                        mon_sp := "XV_ERRORMON_TIME",
                        "open/close" => "H/SSR_019_XV12_OPEN",
                        fault => "H/SSR_019_XV12_Faulty",
                        status => "H/SSR_019_XV12_Status");
       "H/SSR_019_XV13"("A/M" := "H/SSR_019_AM",   // "valve"
                        open_auto := "H/SSR_019_XV13_CMD",
                        open_man := "H/SSR_019_XV13_MCMD",
                        fbk_open := "SIM_VALVE"."H/SSR_019_XV13_OPENFB",
                        fbk_close := "SIM_VALVE"."H/SSR_019_XV13_CLOSEFB",
                        reset := "H/SSR_019_XV13_RESET",
                        intl := 1,
                        Mon_En := 1,
                        mon_sp := "XV_ERRORMON_TIME",
                        "open/close" => "H/SSR_019_XV13_OPEN",
                        fault => "H/SSR_019_XV13_Faulty",
                        status => "H/SSR_019_XV13_Status");
   END_IF;
END_REGION

REGION Network 6: AI_H/SSR_019_ Reading
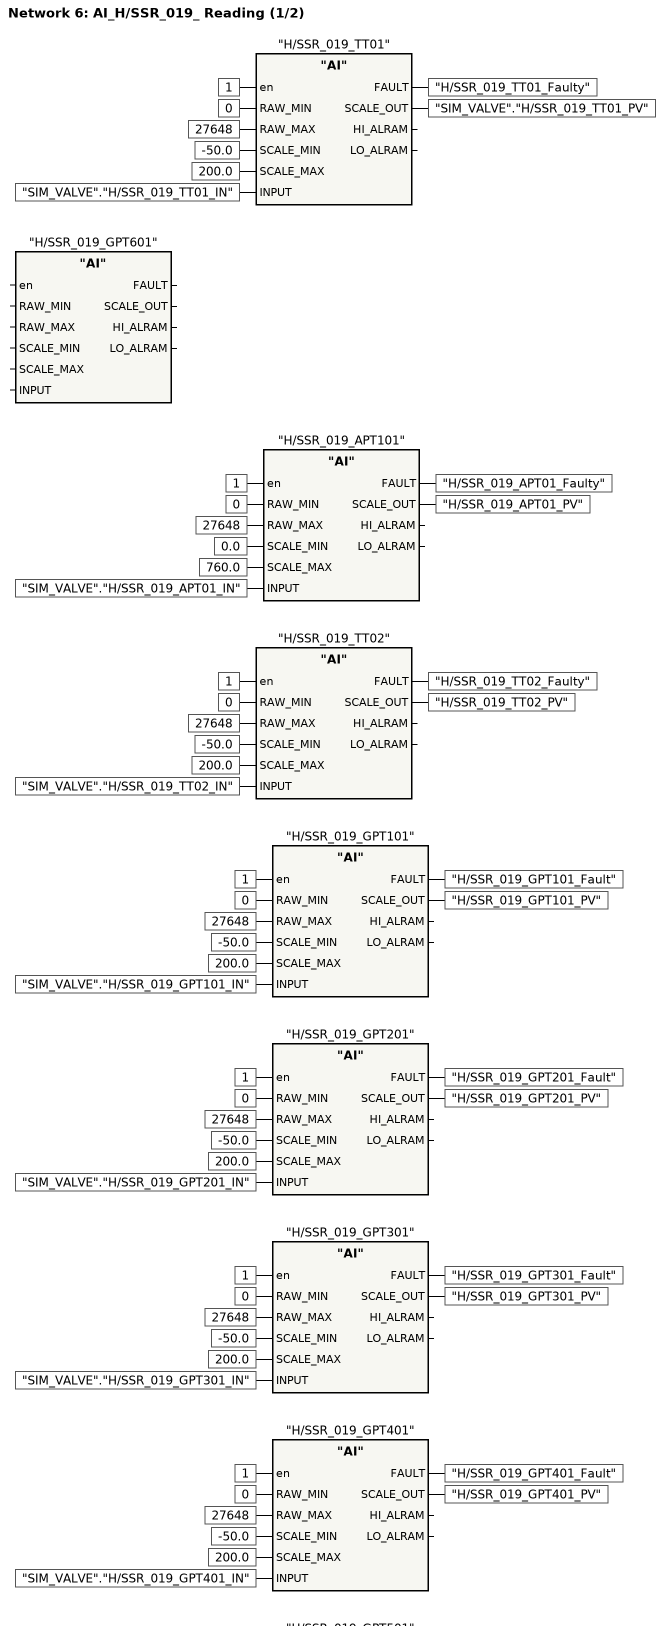
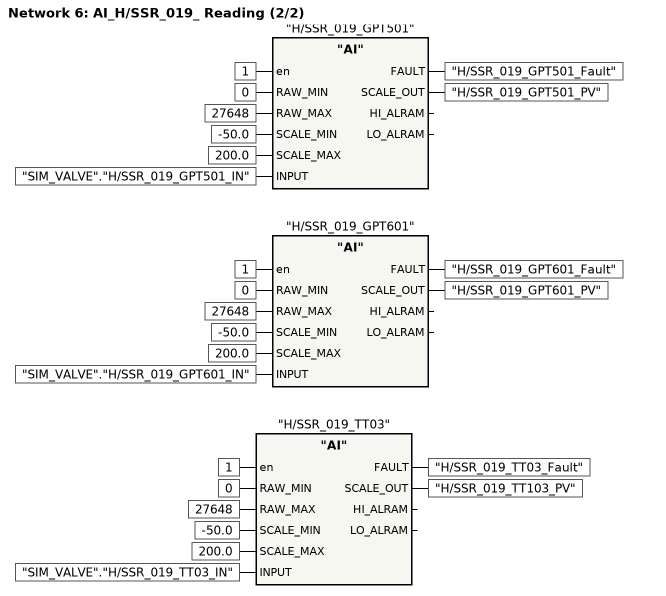
   IF 1 THEN
       "H/SSR_019_TT01"(RAW_MIN := 0,   // "AI"
                        RAW_MAX := 27648,
                        SCALE_MIN := -50.0,
                        SCALE_MAX := 200.0,
                        INPUT := "SIM_VALVE"."H/SSR_019_TT01_IN",
                        FAULT => "H/SSR_019_TT01_Faulty",
                        SCALE_OUT => "SIM_VALVE"."H/SSR_019_TT01_PV");
   END_IF;
   "H/SSR_019_GPT601"();   // "AI"
   IF 1 THEN
       "H/SSR_019_APT101"(RAW_MIN := 0,   // "AI"
                          RAW_MAX := 27648,
                          SCALE_MIN := 0.0,
                          SCALE_MAX := 760.0,
                          INPUT := "SIM_VALVE"."H/SSR_019_APT01_IN",
                          FAULT => "H/SSR_019_APT01_Faulty",
                          SCALE_OUT => "H/SSR_019_APT01_PV");
       "H/SSR_019_TT02"(RAW_MIN := 0,   // "AI"
                        RAW_MAX := 27648,
                        SCALE_MIN := -50.0,
                        SCALE_MAX := 200.0,
                        INPUT := "SIM_VALVE"."H/SSR_019_TT02_IN",
                        FAULT => "H/SSR_019_TT02_Faulty",
                        SCALE_OUT => "H/SSR_019_TT02_PV");
       "H/SSR_019_GPT101"(RAW_MIN := 0,   // "AI"
                          RAW_MAX := 27648,
                          SCALE_MIN := -50.0,
                          SCALE_MAX := 200.0,
                          INPUT := "SIM_VALVE"."H/SSR_019_GPT101_IN",
                          FAULT => "H/SSR_019_GPT101_Fault",
                          SCALE_OUT => "H/SSR_019_GPT101_PV");
       "H/SSR_019_GPT201"(RAW_MIN := 0,   // "AI"
                          RAW_MAX := 27648,
                          SCALE_MIN := -50.0,
                          SCALE_MAX := 200.0,
                          INPUT := "SIM_VALVE"."H/SSR_019_GPT201_IN",
                          FAULT => "H/SSR_019_GPT201_Fault",
                          SCALE_OUT => "H/SSR_019_GPT201_PV");
       "H/SSR_019_GPT301"(RAW_MIN := 0,   // "AI"
                          RAW_MAX := 27648,
                          SCALE_MIN := -50.0,
                          SCALE_MAX := 200.0,
                          INPUT := "SIM_VALVE"."H/SSR_019_GPT301_IN",
                          FAULT => "H/SSR_019_GPT301_Fault",
                          SCALE_OUT => "H/SSR_019_GPT301_PV");
       "H/SSR_019_GPT401"(RAW_MIN := 0,   // "AI"
                          RAW_MAX := 27648,
                          SCALE_MIN := -50.0,
                          SCALE_MAX := 200.0,
                          INPUT := "SIM_VALVE"."H/SSR_019_GPT401_IN",
                          FAULT => "H/SSR_019_GPT401_Fault",
                          SCALE_OUT => "H/SSR_019_GPT401_PV");
       "H/SSR_019_GPT501"(RAW_MIN := 0,   // "AI"
                          RAW_MAX := 27648,
                          SCALE_MIN := -50.0,
                          SCALE_MAX := 200.0,
                          INPUT := "SIM_VALVE"."H/SSR_019_GPT501_IN",
                          FAULT => "H/SSR_019_GPT501_Fault",
                          SCALE_OUT => "H/SSR_019_GPT501_PV");
       "H/SSR_019_GPT601"(RAW_MIN := 0,   // "AI"
                          RAW_MAX := 27648,
                          SCALE_MIN := -50.0,
                          SCALE_MAX := 200.0,
                          INPUT := "SIM_VALVE"."H/SSR_019_GPT601_IN",
                          FAULT => "H/SSR_019_GPT601_Fault",
                          SCALE_OUT => "H/SSR_019_GPT601_PV");
       "H/SSR_019_TT03"(RAW_MIN := 0,   // "AI"
                        RAW_MAX := 27648,
                        SCALE_MIN := -50.0,
                        SCALE_MAX := 200.0,
                        INPUT := "SIM_VALVE"."H/SSR_019_TT03_IN",
                        FAULT => "H/SSR_019_TT03_Fault",
                        SCALE_OUT => "H/SSR_019_TT103_PV");
   END_IF;
END_REGION

REGION Network 7: Agitaor
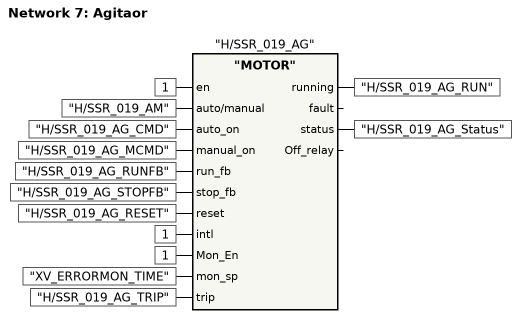
   IF 1 THEN
       "H/SSR_019_AG"("auto/manual" := "H/SSR_019_AM",   // "MOTOR"
                      auto_on := "H/SSR_019_AG_CMD",
                      manual_on := "H/SSR_019_AG_MCMD",
                      run_fb := "H/SSR_019_AG_RUNFB",
                      stop_fb := "H/SSR_019_AG_STOPFB",
                      reset := "H/SSR_019_AG_RESET",
                      intl := 1,
                      Mon_En := 1,
                      mon_sp := "XV_ERRORMON_TIME",
                      trip := "H/SSR_019_AG_TRIP",
                      running => "H/SSR_019_AG_RUN",
                      status => "H/SSR_019_AG_Status");
   END_IF;
END_REGION

REGION Network 8: H/SSR_019 GLOBAL RESET
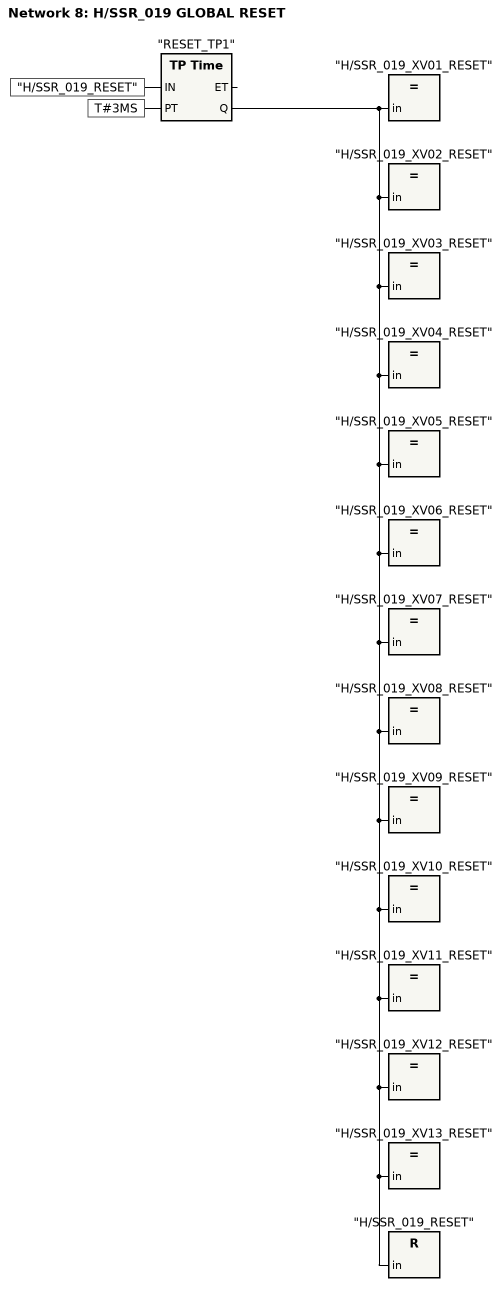
   "RESET_TP1".TP(IN := "H/SSR_019_RESET", PT := T#3MS);
   "H/SSR_019_XV01_RESET" := "RESET_TP1".Q;
   "H/SSR_019_XV02_RESET" := "RESET_TP1".Q;
   "H/SSR_019_XV03_RESET" := "RESET_TP1".Q;
   "H/SSR_019_XV04_RESET" := "RESET_TP1".Q;
   "H/SSR_019_XV05_RESET" := "RESET_TP1".Q;
   "H/SSR_019_XV06_RESET" := "RESET_TP1".Q;
   "H/SSR_019_XV07_RESET" := "RESET_TP1".Q;
   "H/SSR_019_XV08_RESET" := "RESET_TP1".Q;
   "H/SSR_019_XV09_RESET" := "RESET_TP1".Q;
   "H/SSR_019_XV10_RESET" := "RESET_TP1".Q;
   "H/SSR_019_XV11_RESET" := "RESET_TP1".Q;
   "H/SSR_019_XV12_RESET" := "RESET_TP1".Q;
   "H/SSR_019_XV13_RESET" := "RESET_TP1".Q;
   IF "RESET_TP1".Q THEN "H/SSR_019_RESET" := FALSE; END_IF;
END_REGION

REGION Network 9: HOOTER
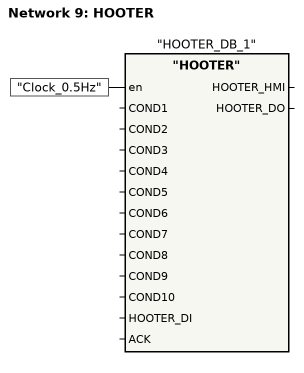
   IF "Clock_0.5Hz" THEN
       "HOOTER_DB_1"();   // "HOOTER"
   END_IF;
END_REGION
END_ORGANIZATION_BLOCK

FUNCTION_BLOCK "valve"   // FB8, LAD
{ S7_Optimized_Access := 'FALSE' }
VERSION : 0.1
// stored: AutoNumber true, IsIECCheckEnabled false, SetENOAutomatically false, UDAEnableTagReadback false
   VAR_INPUT
      "A/M" : Bool;
      open_auto : Bool;
      open_man : Bool;
      fbk_open : Bool;
      fbk_close : Bool;
      reset : Bool;
      intl : Bool;
      Mon_En : Bool;
      mon_sp : Time;
      run_fb : Bool;
      stop_fb : Bool;
   END_VAR
   VAR_OUTPUT
      "open/close" : Bool;
      fault : Bool;
      status : Int;
   END_VAR
   VAR DB_SPECIFIC
      open_fault : Bool;
      close_fault : Bool;
      IEC_Timer_0_Instance { S7_SetPoint := 'True'} : TON_TIME;
      IEC_Timer_0_Instance_1 { S7_SetPoint := 'True'} : TON_TIME;
      mon : Int;
      pulse : Bool;
      pulse1 : Bool;
      mon1 : Int;
      IEC_Timer_0_Instance_2 { S7_SetPoint := 'True'} : TON_TIME;
   END_VAR
   VAR_TEMP   // added for the SCL form of the ladder/FBD networks
      _w1 : Bool;
   END_VAR
BEGIN

REGION Network 1
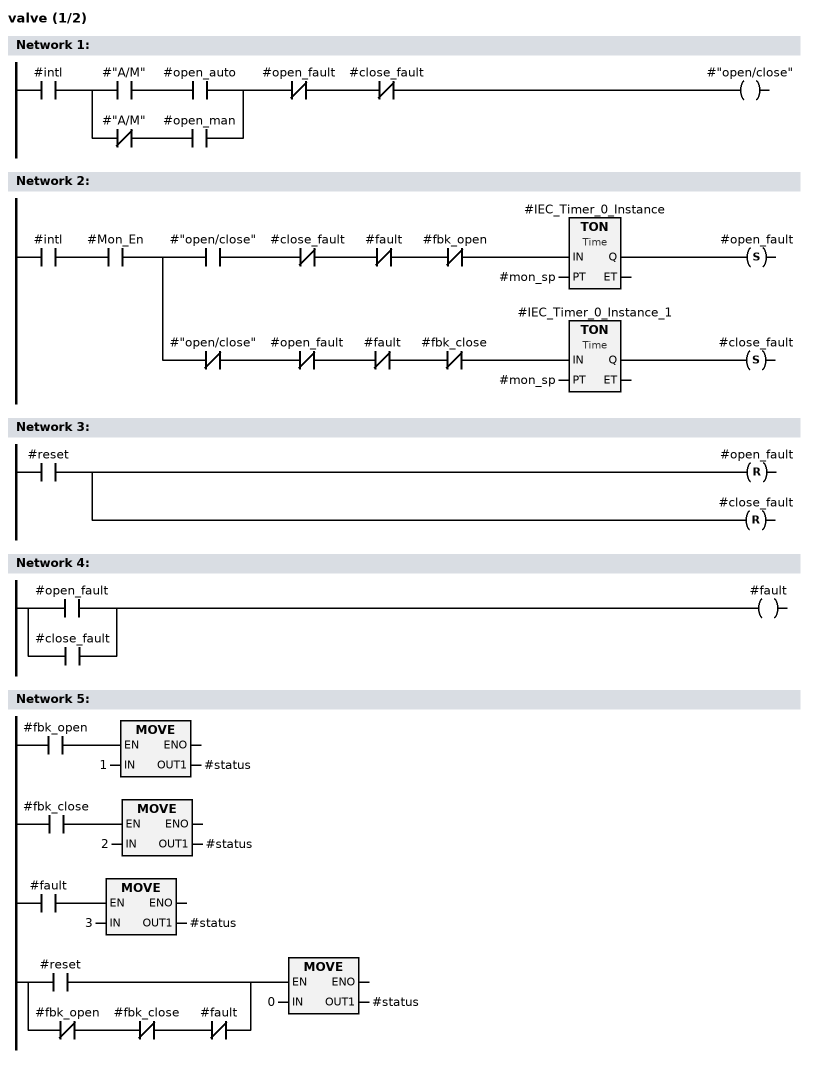
   RUNG wire#powerrail
      Contact( #intl )
      wire#w1
      Contact( #"A/M" )
      Contact( #open_auto )
      wire#w2
      I_Contact( #open_fault )
      I_Contact( #close_fault )
      Coil( #"open/close" )
   END_RUNG
   RUNG wire#w1
      I_Contact( #"A/M" )
      Contact( #open_man )
   END_RUNG wire#w2
   // the same network as SCL:
   #"open/close" := #intl AND ((#"A/M" AND #open_auto) OR (NOT #"A/M" AND #open_man)) AND NOT #open_fault AND NOT #close_fault;
END_REGION

REGION Network 2
   RUNG wire#powerrail
      Contact( #intl )
      Contact( #Mon_En )
      wire#w1
      Contact( #"open/close" )
      I_Contact( #close_fault )
      I_Contact( #fault )
      I_Contact( #fbk_open )
      { S7_Templates := "time_type := Time" } #IEC_Timer_0_Instance.TON(pt := #mon_sp, et =>)
      S_Coil( #open_fault )
   END_RUNG
   RUNG wire#w1
      I_Contact( #"open/close" )
      I_Contact( #open_fault )
      I_Contact( #fault )
      I_Contact( #fbk_close )
      { S7_Templates := "time_type := Time" } #IEC_Timer_0_Instance_1.TON(pt := #mon_sp, et =>)
      S_Coil( #close_fault )
   END_RUNG
   // the same network as SCL:
   #_w1 := #intl AND #Mon_En;
   #IEC_Timer_0_Instance(IN := #_w1 AND #"open/close" AND NOT #close_fault AND NOT #fault AND NOT #fbk_open,   // TON
                         PT := #mon_sp);
   IF #IEC_Timer_0_Instance.Q THEN #open_fault := TRUE; END_IF;
   #IEC_Timer_0_Instance_1(IN := #_w1 AND NOT #"open/close" AND NOT #open_fault AND NOT #fault AND NOT #fbk_close,   // TON
                           PT := #mon_sp);
   IF #IEC_Timer_0_Instance_1.Q THEN #close_fault := TRUE; END_IF;
END_REGION

REGION Network 3
   RUNG wire#powerrail
      Contact( #reset )
      wire#w1
      R_Coil( #open_fault )
   END_RUNG
   RUNG wire#w1
      R_Coil( #close_fault )
   END_RUNG
   // the same network as SCL:
   IF #reset THEN
       #open_fault := FALSE;
       #close_fault := FALSE;
   END_IF;
END_REGION

REGION Network 4
   RUNG wire#powerrail
      Contact( #open_fault )
      wire#w1
      Coil( #fault )
   END_RUNG
   RUNG wire#powerrail
      Contact( #close_fault )
   END_RUNG wire#w1
   // the same network as SCL:
   #fault := #open_fault OR #close_fault;
END_REGION

REGION Network 5
   RUNG wire#powerrail
      Contact( #fbk_open )
      Move(in := 1, out1 => #status)
   END_RUNG
   RUNG wire#powerrail
      Contact( #fbk_close )
      Move(in := 2, out1 => #status)
   END_RUNG
   RUNG wire#powerrail
      Contact( #fault )
      Move(in := 3, out1 => #status)
   END_RUNG
   RUNG wire#powerrail
      Contact( #reset )
      wire#w1
      Move(in := 0, out1 => #status)
   END_RUNG
   RUNG wire#powerrail
      I_Contact( #fbk_open )
      I_Contact( #fbk_close )
      I_Contact( #fault )
   END_RUNG wire#w1
   // the same network as SCL:
   IF #fbk_open THEN #status := 1; END_IF;
   IF #fbk_close THEN #status := 2; END_IF;
   IF #fault THEN #status := 3; END_IF;
   IF #reset OR (NOT #fbk_open AND NOT #fbk_close AND NOT #fault) THEN #status := 0; END_IF;
END_REGION

REGION Network 7
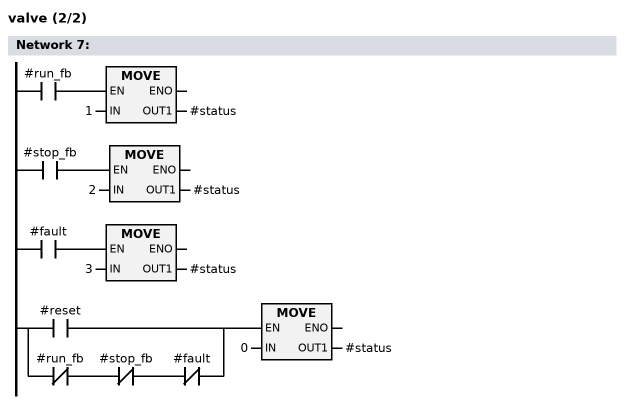
   RUNG wire#powerrail
      Contact( #run_fb )
      Move(in := 1, out1 => #status)
   END_RUNG
   RUNG wire#powerrail
      Contact( #stop_fb )
      Move(in := 2, out1 => #status)
   END_RUNG
   RUNG wire#powerrail
      Contact( #fault )
      Move(in := 3, out1 => #status)
   END_RUNG
   RUNG wire#powerrail
      Contact( #reset )
      wire#w1
      Move(in := 0, out1 => #status)
   END_RUNG
   RUNG wire#powerrail
      I_Contact( #run_fb )
      I_Contact( #stop_fb )
      I_Contact( #fault )
   END_RUNG wire#w1
   // the same network as SCL:
   IF #run_fb THEN #status := 1; END_IF;
   IF #stop_fb THEN #status := 2; END_IF;
   IF #fault THEN #status := 3; END_IF;
   IF #reset OR (NOT #run_fb AND NOT #stop_fb AND NOT #fault) THEN #status := 0; END_IF;
END_REGION
END_FUNCTION_BLOCK

FUNCTION_BLOCK "AI"   // FB3, LAD
{ S7_Optimized_Access := 'TRUE' }
VERSION : 0.1
// stored: AutoNumber true, IsIECCheckEnabled false, IsRetainMemResEnabled false, MemoryReserve 100, SetENOAutomatically false, UDAEnableTagReadback false
   VAR_INPUT
      RAW_MIN : Int;
      RAW_MAX : Int;
      SCALE_MIN : Real;
      SCALE_MAX : Real;
      INPUT : Int;
   END_VAR
   VAR_OUTPUT
      FAULT : Bool;
      SCALE_OUT : Real;
      HI_ALRAM : Bool;
      LO_ALRAM : Bool;
   END_VAR
   VAR
      AI { S7_SetPoint := 'True'} : "SCALING";
      MAX_VALUE { S7_SetPoint := 'True'} : Int;
   END_VAR
BEGIN

REGION Network 1 (SCL)

   IF #INPUT < -100 OR  #INPUT > 27648 THEN
       #FAULT :=1;
   ELSE
       #FAULT := 0;
   END_IF;
   IF NOT #FAULT THEN
       #AI(RAW_MIN := #RAW_MIN,
           RAW_MAX := #RAW_MAX,
           INPUT := #INPUT,
           SCALE_MIN := #SCALE_MIN,
           SCALE_MAX := #SCALE_MAX,
           SCALE_OUT => #SCALE_OUT);
   ELSE
       #SCALE_OUT := 0.0;

   END_IF;
       IF #INPUT < 0 THEN
           #LO_ALRAM := 1;
       ELSE
           #LO_ALRAM := 0;
       END_IF;
       IF #INPUT>27648 THEN
           #HI_ALRAM := 1;
       ELSE
           #HI_ALRAM := 0;

        END_IF;
END_REGION
END_FUNCTION_BLOCK

FUNCTION_BLOCK "SCALING"   // FB4, LAD
{ S7_Optimized_Access := 'TRUE' }
VERSION : 0.1
// stored: AutoNumber true, IsIECCheckEnabled false, IsRetainMemResEnabled false, MemoryReserve 100, SetENOAutomatically false, UDAEnableTagReadback false
   VAR_INPUT
      RAW_MIN : Int;
      RAW_MAX : Int;
      INPUT : Int;
      SCALE_MIN : Real;
      SCALE_MAX : Real;
   END_VAR
   VAR_OUTPUT
      SCALE_OUT : Real;
   END_VAR
   VAR
      TEMP : Real;
   END_VAR
BEGIN

REGION Network 1: SCALING_BLOCK
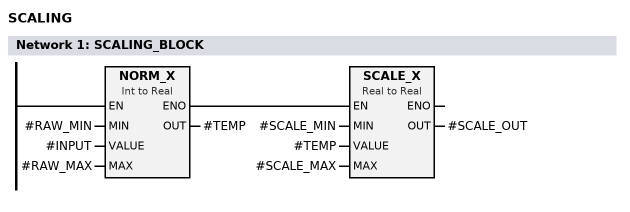
   RUNG wire#powerrail
      { S7_Templates := "[SrcType := Int, DestType := Real]" } Normalize(min := #RAW_MIN, value := #INPUT, max := #RAW_MAX, out => #TEMP)
      { S7_Templates := "[SrcType := Real, DestType := Real]" } Scale(min := #SCALE_MIN, value := #TEMP, max := #SCALE_MAX, out => #SCALE_OUT)
   END_RUNG
   // the same network as SCL:
   #TEMP := NORM_X(MIN := #RAW_MIN, VALUE := #INPUT, MAX := #RAW_MAX);
   #SCALE_OUT := SCALE_X(MIN := #SCALE_MIN, VALUE := #TEMP, MAX := #SCALE_MAX);
END_REGION
END_FUNCTION_BLOCK

FUNCTION_BLOCK "MOTOR"   // FB17, LAD
{ S7_Optimized_Access := 'TRUE' }
VERSION : 0.1
// stored: AutoNumber true, IsIECCheckEnabled false, IsRetainMemResEnabled false, MemoryReserve 100, SetENOAutomatically false, UDAEnableTagReadback false
   VAR_INPUT
      "auto/manual" : Bool;
      auto_on : Bool;
      manual_on : Bool;
      run_fb : Bool;
      stop_fb : Bool;
      reset : Bool;
      intl : Bool;
      Mon_En : Bool;
      mon_sp : Time;
      trip : Bool;
   END_VAR
   VAR_OUTPUT
      running : Bool;
      fault : Bool;
      status : Int;
      Off_relay : Bool;
   END_VAR
   VAR
      on_fault : Bool;
      off_fault : Bool;
      IEC_Timer_0_Instance : TON_TIME;
      IEC_Timer_0_Instance_1 { S7_SetPoint := 'True'} : TON_TIME;
      mon { S7_SetPoint := 'True'} : Int;
      pulse : Bool;
      pulse1 : Bool;
      mon1 : Int;
      IEC_Timer_0_Instance_2 : TON_TIME;
      off_pls : Bool;
      Off_relay_bit : Bool;
      timer1 { S7_SetPoint := 'True'} : TON_TIME;
   END_VAR
   VAR_TEMP   // added for the SCL form of the ladder/FBD networks
      _w1 : Bool;
      _w2 : Bool;
   END_VAR
BEGIN

REGION Network 1
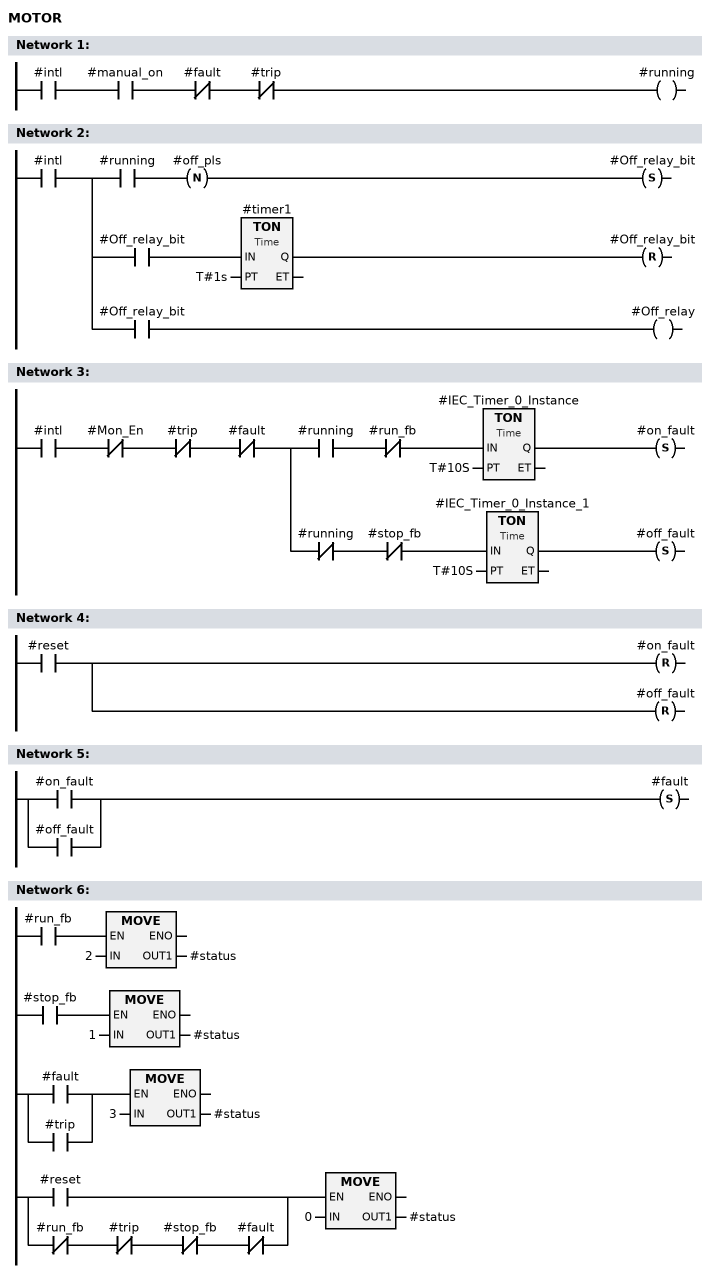
   RUNG wire#powerrail
      Contact( #intl )
      Contact( #manual_on )
      I_Contact( #fault )
      I_Contact( #trip )
      Coil( #running )
   END_RUNG
   // the same network as SCL:
   #running := #intl AND #manual_on AND NOT #fault AND NOT #trip;
END_REGION

REGION Network 2
   RUNG wire#powerrail
      Contact( #intl )
      wire#w1
      Contact( #running )
      N_Trig( #off_pls )
      S_Coil( #Off_relay_bit )
   END_RUNG
   RUNG wire#w1
      Contact( #Off_relay_bit )
      { S7_Templates := "time_type := Time" } #timer1.TON(pt := T#1s, et =>)
      R_Coil( #Off_relay_bit )
   END_RUNG
   RUNG wire#w1
      Contact( #Off_relay_bit )
      Coil( #Off_relay )
   END_RUNG
   // the same network as SCL:
   #_w1 := #intl AND #running;
   #_w2 := NOT #_w1 AND #off_pls;   // falling edge
   #off_pls := #_w1;
   IF #_w2 THEN #Off_relay_bit := TRUE; END_IF;
   #timer1(IN := #intl AND #Off_relay_bit, PT := T#1s);   // TON
   IF #timer1.Q THEN #Off_relay_bit := FALSE; END_IF;
   #Off_relay := #intl AND #Off_relay_bit;
END_REGION

REGION Network 3
   RUNG wire#powerrail
      Contact( #intl )
      I_Contact( #Mon_En )
      I_Contact( #trip )
      I_Contact( #fault )
      wire#w1
      Contact( #running )
      I_Contact( #run_fb )
      { S7_Templates := "time_type := Time" } #IEC_Timer_0_Instance.TON(pt := T#10S, et =>)
      S_Coil( #on_fault )
   END_RUNG
   RUNG wire#w1
      I_Contact( #running )
      I_Contact( #stop_fb )
      { S7_Templates := "time_type := Time" } #IEC_Timer_0_Instance_1.TON(pt := T#10S, et =>)
      S_Coil( #off_fault )
   END_RUNG
   // the same network as SCL:
   #_w1 := #intl AND NOT #Mon_En AND NOT #trip AND NOT #fault;
   #IEC_Timer_0_Instance(IN := #_w1 AND #running AND NOT #run_fb, PT := T#10S);   // TON
   IF #IEC_Timer_0_Instance.Q THEN #on_fault := TRUE; END_IF;
   #IEC_Timer_0_Instance_1(IN := #_w1 AND NOT #running AND NOT #stop_fb, PT := T#10S);   // TON
   IF #IEC_Timer_0_Instance_1.Q THEN #off_fault := TRUE; END_IF;
END_REGION

REGION Network 4
   RUNG wire#powerrail
      Contact( #reset )
      wire#w1
      R_Coil( #on_fault )
   END_RUNG
   RUNG wire#w1
      R_Coil( #off_fault )
   END_RUNG
   // the same network as SCL:
   IF #reset THEN
       #on_fault := FALSE;
       #off_fault := FALSE;
   END_IF;
END_REGION

REGION Network 5
   RUNG wire#powerrail
      Contact( #on_fault )
      wire#w1
      S_Coil( #fault )
   END_RUNG
   RUNG wire#powerrail
      Contact( #off_fault )
   END_RUNG wire#w1
   // the same network as SCL:
   IF #on_fault OR #off_fault THEN #fault := TRUE; END_IF;
END_REGION

REGION Network 6
   RUNG wire#powerrail
      Contact( #run_fb )
      Move(in := 2, out1 => #status)
   END_RUNG
   RUNG wire#powerrail
      Contact( #stop_fb )
      Move(in := 1, out1 => #status)
   END_RUNG
   RUNG wire#powerrail
      Contact( #fault )
      wire#w1
      Move(in := 3, out1 => #status)
   END_RUNG
   RUNG wire#powerrail
      Contact( #trip )
   END_RUNG wire#w1
   RUNG wire#powerrail
      Contact( #reset )
      wire#w2
      Move(in := 0, out1 => #status)
   END_RUNG
   RUNG wire#powerrail
      I_Contact( #run_fb )
      I_Contact( #trip )
      I_Contact( #stop_fb )
      I_Contact( #fault )
   END_RUNG wire#w2
   // the same network as SCL:
   IF #run_fb THEN #status := 2; END_IF;
   IF #stop_fb THEN #status := 1; END_IF;
   IF #fault OR #trip THEN #status := 3; END_IF;
   IF #reset OR (NOT #run_fb AND NOT #trip AND NOT #stop_fb AND NOT #fault) THEN #status := 0; END_IF;
END_REGION
END_FUNCTION_BLOCK

FUNCTION_BLOCK "HOOTER"   // FB5, FBD
{ S7_Optimized_Access := 'TRUE' }
VERSION : 0.1
// stored: AutoNumber true, IsIECCheckEnabled false, IsRetainMemResEnabled false, MemoryReserve 100, SetENOAutomatically false, UDAEnableTagReadback false
   VAR_INPUT
      COND1 : Bool;
      COND2 : Bool;
      COND3 : Bool;
      COND4 : Bool;
      COND5 : Bool;
      COND6 : Bool;
      COND7 : Bool;
      COND8 : Bool;
      COND9 : Bool;
      COND10 : Bool;
      HOOTER_DI : Bool;
   END_VAR
   VAR_OUTPUT
      HOOTER_HMI : Bool;
      HOOTER_DO : Bool;
   END_VAR
   VAR_IN_OUT
      ACK : Bool;
   END_VAR
   VAR
      RS1 : Bool;
      RS2 : Bool;
      RS3 : Bool;
      RS4 : Bool;
      RS5 : Bool;
      RS6 : Bool;
      RS7 : Bool;
      RS8 : Bool;
      RS9 : Bool;
      RS10 : Bool;
   END_VAR
BEGIN

REGION Network 1
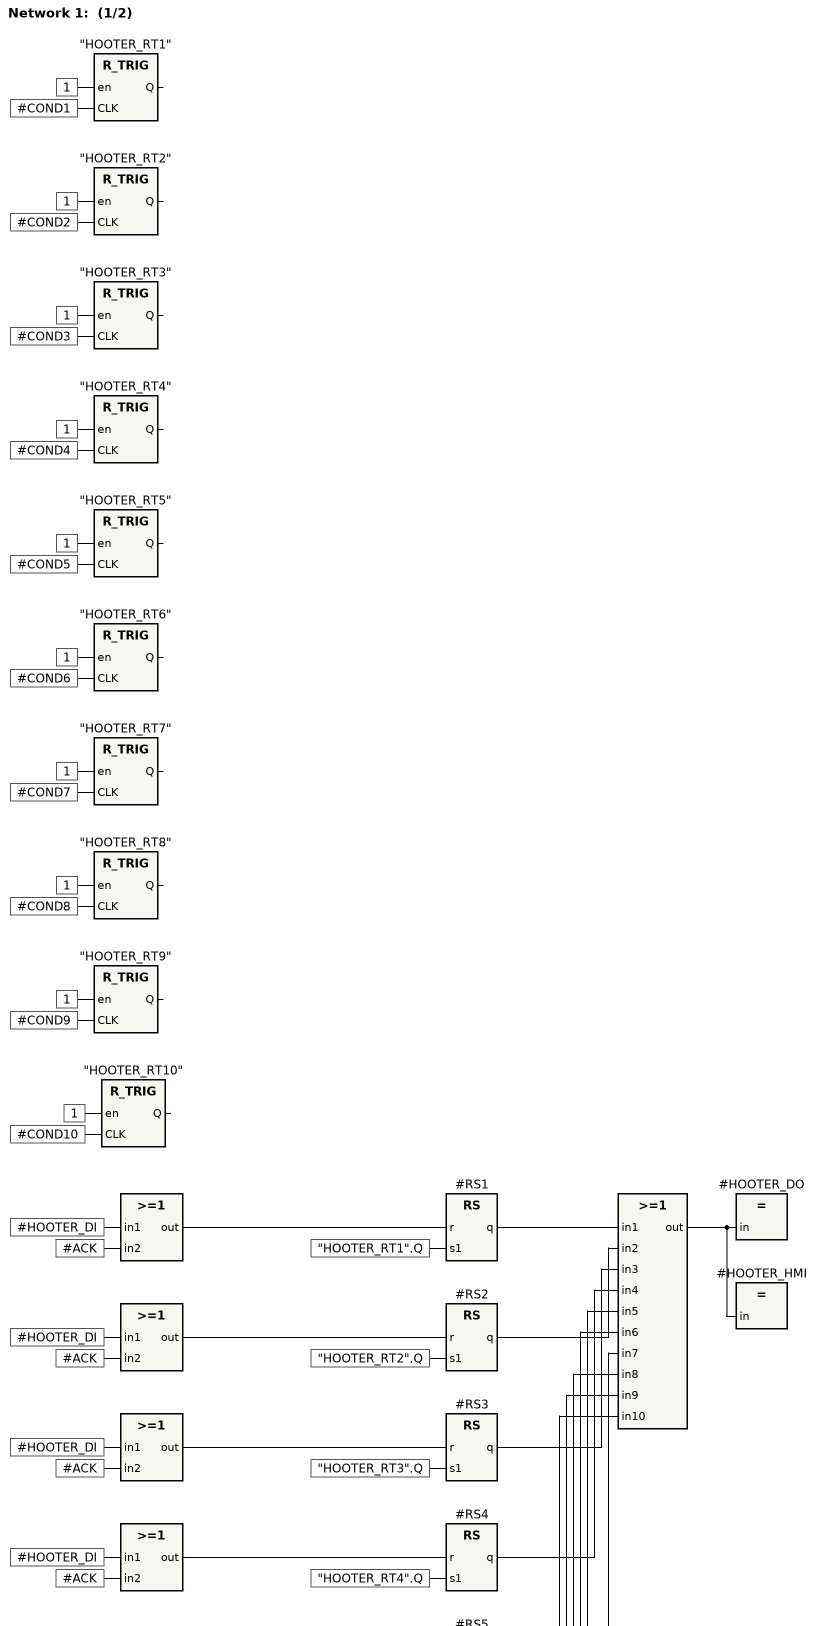
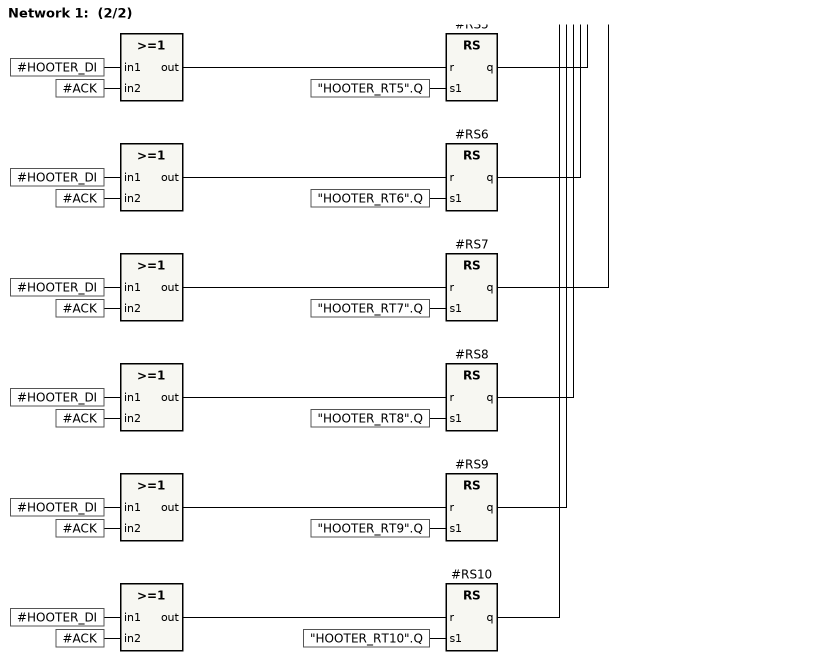
   IF 1 THEN
       "HOOTER_RT1"(CLK := #COND1);   // R_TRIG
       "HOOTER_RT2"(CLK := #COND2);   // R_TRIG
       "HOOTER_RT3"(CLK := #COND3);   // R_TRIG
       "HOOTER_RT4"(CLK := #COND4);   // R_TRIG
       "HOOTER_RT5"(CLK := #COND5);   // R_TRIG
       "HOOTER_RT6"(CLK := #COND6);   // R_TRIG
       "HOOTER_RT7"(CLK := #COND7);   // R_TRIG
       "HOOTER_RT8"(CLK := #COND8);   // R_TRIG
       "HOOTER_RT9"(CLK := #COND9);   // R_TRIG
       "HOOTER_RT10"(CLK := #COND10);   // R_TRIG
   END_IF;
   IF #HOOTER_DI OR #ACK THEN
       #RS1 := FALSE;   // RS flip-flop
   END_IF;
   IF "HOOTER_RT1".Q THEN #RS1 := TRUE; END_IF;
   IF #HOOTER_DI OR #ACK THEN
       #RS2 := FALSE;   // RS flip-flop
   END_IF;
   IF "HOOTER_RT2".Q THEN #RS2 := TRUE; END_IF;
   IF #HOOTER_DI OR #ACK THEN
       #RS3 := FALSE;   // RS flip-flop
   END_IF;
   IF "HOOTER_RT3".Q THEN #RS3 := TRUE; END_IF;
   IF #HOOTER_DI OR #ACK THEN
       #RS4 := FALSE;   // RS flip-flop
   END_IF;
   IF "HOOTER_RT4".Q THEN #RS4 := TRUE; END_IF;
   IF #HOOTER_DI OR #ACK THEN
       #RS5 := FALSE;   // RS flip-flop
   END_IF;
   IF "HOOTER_RT5".Q THEN #RS5 := TRUE; END_IF;
   IF #HOOTER_DI OR #ACK THEN
       #RS6 := FALSE;   // RS flip-flop
   END_IF;
   IF "HOOTER_RT6".Q THEN #RS6 := TRUE; END_IF;
   IF #HOOTER_DI OR #ACK THEN
       #RS7 := FALSE;   // RS flip-flop
   END_IF;
   IF "HOOTER_RT7".Q THEN #RS7 := TRUE; END_IF;
   IF #HOOTER_DI OR #ACK THEN
       #RS8 := FALSE;   // RS flip-flop
   END_IF;
   IF "HOOTER_RT8".Q THEN #RS8 := TRUE; END_IF;
   IF #HOOTER_DI OR #ACK THEN
       #RS9 := FALSE;   // RS flip-flop
   END_IF;
   IF "HOOTER_RT9".Q THEN #RS9 := TRUE; END_IF;
   IF #HOOTER_DI OR #ACK THEN
       #RS10 := FALSE;   // RS flip-flop
   END_IF;
   IF "HOOTER_RT10".Q THEN #RS10 := TRUE; END_IF;
   #HOOTER_DO := #RS1 OR #RS2 OR #RS3 OR #RS4 OR #RS5 OR #RS6 OR #RS7 OR #RS8 OR #RS9 OR #RS10;
   #HOOTER_HMI := #HOOTER_DO;
END_REGION
END_FUNCTION_BLOCK

ORGANIZATION_BLOCK "PID Cyclic interrupt"   // OB30, FBD, CyclicInterrupt
{ S7_Optimized_Access := 'TRUE' }
VERSION : 0.1
// stored: AutoNumber true, IsIECCheckEnabled false, SetENOAutomatically false
   VAR_INPUT
      Initial_Call : Bool;   // Initial call of this OB
      Event_Count : Int;   // Events discarded
   END_VAR
BEGIN

REGION Network 1: Utility_PID
   // Utility_PID
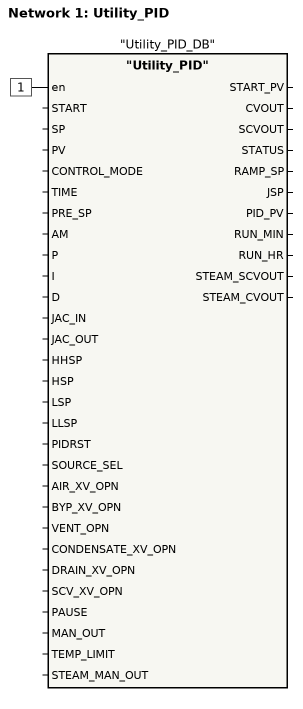
   IF 1 THEN
       "Utility_PID_DB"();   // "Utility_PID"
   END_IF;
END_REGION
END_ORGANIZATION_BLOCK

FUNCTION_BLOCK "Utility_PID"   // FB2, FBD
TITLE = Utility PID Control
{ S7_Optimized_Access := 'TRUE' }
VERSION : 0.1
// Utility PID Control
// stored: AutoNumber true, IsIECCheckEnabled false, IsRetainMemResEnabled false, MemoryReserve 100, SetENOAutomatically false, UDAEnableTagReadback false
   VAR_INPUT
      START : Bool;
      SP : Real;
      PV : Real;
      CONTROL_MODE : Int;
      "TIME" : Int;
      PRE_SP : Int;
      AM : Bool;
      P : Int;
      I : Int;
      D : Int;
      JAC_IN : Real;
      JAC_OUT : Real;
      HHSP : Real;
      HSP : Real;
      LSP : Real;
      LLSP : Real;
      PIDRST : Bool;
      SOURCE_SEL : Int;
      AIR_XV_OPN : Bool;
      BYP_XV_OPN : Bool;
      VENT_OPN : Bool;
      CONDENSATE_XV_OPN : Bool;
      DRAIN_XV_OPN : Bool;
      SCV_XV_OPN : Bool;
   END_VAR
   VAR_OUTPUT
      START_PV : Real;
      CVOUT : Int;
      SCVOUT : Real;
      STATUS : Int;
      RAMP_SP : Real;
      JSP : Real;
      PID_PV : Real;
      RUN_MIN : Int;
      RUN_HR : Int;
      STEAM_SCVOUT : Real;
      STEAM_CVOUT : Int;
   END_VAR
   VAR_IN_OUT
      PAUSE : Bool;
      MAN_OUT : Real;
      TEMP_LIMIT : Real;
      STEAM_MAN_OUT : Real;
   END_VAR
   VAR
      RAMP_MODE : Bool;
      MAINT_MODE : Bool;
      J_MAINT_MODE : Bool;
      NO_RAMP : Bool;
      HEAT_COOL : Bool;
      BSTBIT : Bool;
      HOLD : Int;
      RAMP : Real;
      RAMP_RST : Bool;
      RMPSTART : Bool;
      Ramp_Substitute : Real;
      RAMP_INIT_RST : Bool;
      JKT_RAMP : Bool;
      MASS_CONTROL : Bool;
      TIMER_TRIG : Bool;
      iSTEAM_SCVOUT : Real;
      iSTEAM_CVOUT : Int;
      iSTEAM_SCV_SCL : Real;
      iSTEAM_CV_SCL : Int;
      iDRAIN_UP : Bool;
   END_VAR
BEGIN

REGION Network 1: Mode Selection
   // Mode Selection
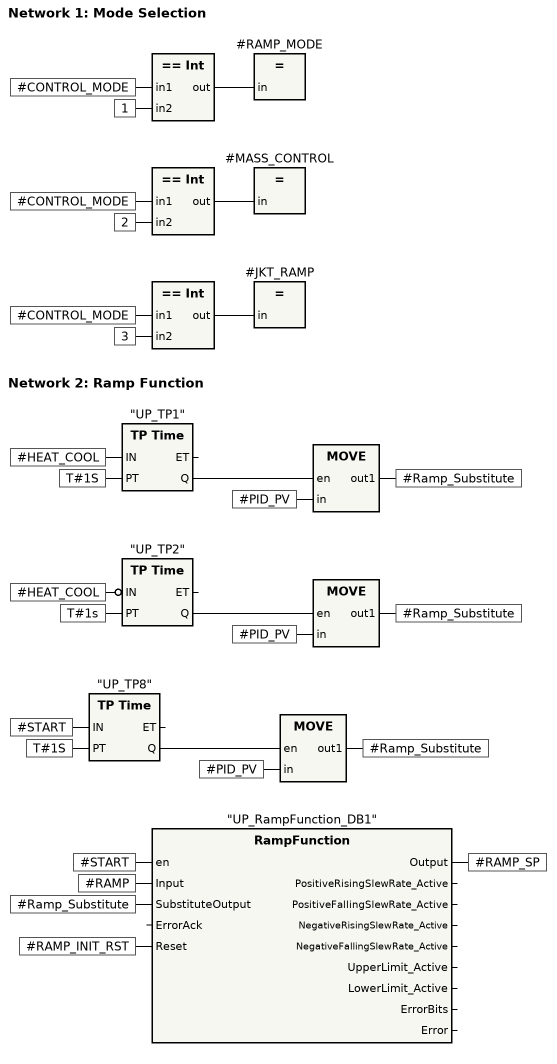
   #RAMP_MODE := #CONTROL_MODE = 1;
   #MASS_CONTROL := #CONTROL_MODE = 2;
   #JKT_RAMP := #CONTROL_MODE = 3;
END_REGION

REGION Network 2: Ramp Function
   // Ramp Function
   "UP_TP1".TP(IN := #HEAT_COOL, PT := T#1S);
   IF "UP_TP1".Q THEN #Ramp_Substitute := #PID_PV; END_IF;
   "UP_TP2".TP(IN := NOT #HEAT_COOL, PT := T#1s);
   IF "UP_TP2".Q THEN #Ramp_Substitute := #PID_PV; END_IF;
   "UP_TP8".TP(IN := #START, PT := T#1S);
   IF "UP_TP8".Q THEN #Ramp_Substitute := #PID_PV; END_IF;
   IF #START THEN
       "UP_RampFunction_DB1"(Input := #RAMP,   // RampFunction
                             SubstituteOutput := #Ramp_Substitute,
                             Reset := #RAMP_INIT_RST,
                             Output => #RAMP_SP);
   END_IF;
END_REGION

REGION Network 3: Ramp Reset
   // Ramp Reset
